C08959=1014.055,42.022,-115.275,165.854,58.897,160.635
C08960=1014.061,42.301,-115.291,165.856,58.886,160.634
C08961=1014.066,42.582,-115.308,165.859,58.876,160.633
C08962=1014.071,42.863,-115.324,165.862,58.866,160.631
C08963=1014.075,43.112,-115.338,165.863,58.857,160.630
C08964=1014.080,43.362,-115.352,165.865,58.848,160.628
C08965=1014.085,43.611,-115.367,165.867,58.838,160.627
C08966=1014.089,43.860,-115.381,165.869,58.829,160.626
C08967=1014.094,44.110,-115.396,165.872,58.820,160.625
C08968=1014.099,44.360,-115.410,165.875,58.810,160.624
C08969=1014.103,44.609,-115.424,165.877,58.800,160.622
C08970=1014.108,44.859,-115.440,165.879,58.791,160.621
C08971=1014.113,45.108,-115.454,165.881,58.782,160.620
C08972=1014.117,45.358,-115.468,165.883,58.773,160.619
C08973=1014.121,45.608,-115.483,165.885,58.763,160.617
C08974=1014.126,45.857,-115.497,165.887,58.754,160.616
C08975=1014.131,46.106,-115.512,165.890,58.745,160.615
C08976=1014.135,46.356,-115.526,165.892,58.735,160.613
C08977=1014.140,46.606,-115.541,165.894,58.726,160.612
C08978=1014.144,46.855,-115.555,165.896,58.716,160.611
C08979=1014.149,47.104,-115.570,165.898,58.707,160.610
C08980=1014.154,47.354,-115.585,165.900,58.697,160.608
C08981=1014.158,47.603,-115.599,165.902,58.688,160.607
C08982=1014.163,47.853,-115.613,165.905,58.678,160.606
C08983=1014.168,48.102,-115.628,165.907,58.668,160.604
C08984=1014.173,48.352,-115.643,165.910,58.659,160.603
C08985=1014.177,48.601,-115.657,165.911,58.650,160.602
C08986=1014.182,48.851,-115.671,165.914,58.641,160.601
C08987=1014.187,49.101,-115.686,165.916,58.631,160.599
C08988=1014.191,49.351,-115.701,165.917,58.621,160.598
C08989=1014.196,49.600,-115.715,165.921,58.612,160.597
C08990=1014.200,49.850,-115.730,165.923,58.602,160.596
C08991=1014.205,50.099,-115.745,165.924,58.592,160.594
C08992=1014.210,50.349,-115.759,165.927,58.583,160.593
C08993=1014.214,50.598,-115.773,165.929,58.573,160.592
C08994=1014.219,50.847,-115.788,165.931,58.564,160.590
C08995=1014.224,51.097,-115.803,165.934,58.554,160.589
C08996=1014.228,51.347,-115.818,165.936,58.544,160.588
C08997=1014.232,51.596,-115.833,165.938,58.535,160.586
C08998=1014.237,51.846,-115.847,165.940,58.525,160.585
C08999=1014.242,52.096,-115.862,165.943,58.515,160.584
C09000=1014.247,52.345,-115.877,165.945,58.506,160.583
C09001=1014.251,52.594,-115.891,165.947,58.496,160.581
C09002=1014.256,52.844,-115.905,165.949,58.486,160.580
C09003=1014.261,53.093,-115.921,165.952,58.477,160.579
C09004=1014.266,53.343,-115.935,165.954,58.467,160.577
C09005=1014.270,53.593,-115.949,165.956,58.457,160.576
C09006=1014.275,53.842,-115.964,165.958,58.448,160.574
C09007=1014.279,54.091,-115.979,165.961,58.437,160.573
C09008=1014.285,54.341,-115.994,165.962,58.428,160.572
C09009=1014.289,54.591,-116.008,165.964,58.418,160.570
C09010=1014.294,54.841,-116.023,165.968,58.409,160.569
C09011=1014.299,55.090,-116.038,165.970,58.399,160.568
C09012=1014.303,55.339,-116.052,165.971,58.389,160.567
C09013=1014.308,55.588,-116.067,165.974,58.379,160.565
C09014=1014.313,55.838,-116.082,165.976,58.369,160.564
C09015=1014.318,56.088,-116.096,165.978,58.359,160.562
C09016=1014.323,56.337,-116.111,165.981,58.349,160.561
C09017=1014.327,56.587,-116.126,165.983,58.340,160.560
C09018=1014.332,56.836,-116.141,165.985,58.330,160.558
C09019=1014.337,57.086,-116.155,165.988,58.320,160.557
C09020=1014.342,57.335,-116.170,165.990,58.310,160.556
C09021=1014.346,57.585,-116.185,165.993,58.300,160.555
C09022=1014.351,57.835,-116.199,165.995,58.290,160.553
C09023=1014.357,58.115,-116.216,165.997,58.279,160.552
C09024=1014.362,58.394,-116.233,166.000,58.268,160.550
C09025=1014.367,58.675,-116.249,166.003,58.257,160.549
C09026=1014.372,58.956,-116.266,166.004,58.245,160.547
C09027=1014.377,59.205,-116.280,166.007,58.235,160.546
C09028=1014.382,59.455,-116.296,166.009,58.226,160.544
C09029=1014.387,59.705,-116.310,166.011,58.216,160.543
C09030=1014.392,59.954,-116.325,166.014,58.206,160.542
C09031=1014.397,60.204,-116.340,166.016,58.196,160.540
C09032=1014.401,60.452,-116.355,166.019,58.186,160.539
C09033=1014.406,60.702,-116.369,166.020,58.176,160.537
C09034=1014.411,60.951,-116.384,166.023,58.165,160.536
C09035=1014.416,61.201,-116.399,166.025,58.156,160.535
C09036=1014.421,61.451,-116.414,166.028,58.146,160.533
C09037=1014.426,61.700,-116.429,166.030,58.136,160.532
C09038=1014.430,61.950,-116.443,166.033,58.126,160.531
C09039=1014.436,62.199,-116.459,166.034,58.115,160.529
C09040=1014.440,62.449,-116.473,166.037,58.105,160.528
C09041=1014.445,62.698,-116.488,166.039,58.096,160.526
C09042=1014.449,62.948,-116.503,166.042,58.085,160.525
C09043=1014.454,63.198,-116.518,166.044,58.076,160.524
C09044=1014.459,63.447,-116.534,166.046,58.066,160.522
C09045=1014.464,63.696,-116.549,166.049,58.056,160.521
C09046=1014.468,63.946,-116.564,166.051,58.046,160.520
C09047=1014.473,64.196,-116.579,166.054,58.036,160.519
C09048=1014.478,64.445,-116.595,166.056,58.026,160.517
C09049=1014.482,64.694,-116.610,166.058,58.016,160.516
C09050=1014.487,64.944,-116.624,166.061,58.006,160.514
C09051=1014.491,65.193,-116.640,166.062,57.996,160.513
C09052=1014.496,65.442,-116.655,166.066,57.986,160.512
C09053=1014.501,65.692,-116.670,166.067,57.977,160.510
C09054=1014.506,65.941,-116.686,166.069,57.967,160.509
C09055=1014.510,66.191,-116.700,166.072,57.956,160.507
C09056=1014.515,66.441,-116.716,166.074,57.946,160.506
C09057=1014.520,66.690,-116.731,166.077,57.936,160.505
C09058=1014.525,66.939,-116.747,166.079,57.927,160.503
C09059=1014.529,67.189,-116.762,166.082,57.917,160.502
C09060=1014.534,67.438,-116.778,166.084,57.907,160.501
C09061=1014.538,67.688,-116.793,166.086,57.896,160.499
C09062=1014.543,67.938,-116.808,166.088,57.886,160.498
C09063=1014.548,68.187,-116.823,166.090,57.877,160.497
C09064=1014.553,68.436,-116.839,166.093,57.867,160.495
C09065=1014.557,68.686,-116.854,166.095,57.857,160.494
C09066=1014.562,68.935,-116.870,166.098,57.846,160.492
C09067=1014.566,69.185,-116.885,166.100,57.837,160.491
C09068=1014.571,69.434,-116.901,166.103,57.827,160.490
C09069=1014.576,69.684,-116.916,166.105,57.817,160.488
C09070=1014.581,69.934,-116.932,166.108,57.807,160.487
C09071=1014.585,70.183,-116.948,166.109,57.796,160.486
C09072=1014.591,70.433,-116.963,166.111,57.787,160.484
C09073=1014.595,70.682,-116.979,166.115,57.777,160.483
C09074=1014.599,70.932,-116.994,166.117,57.767,160.482
C09075=1014.604,71.181,-117.010,166.119,57.756,160.480
C09076=1014.608,71.431,-117.025,166.121,57.747,160.479
C09077=1014.614,71.680,-117.040,166.124,57.737,160.478
C09078=1014.618,71.929,-117.056,166.126,57.727,160.476
C09079=1014.623,72.179,-117.071,166.129,57.716,160.475
C09080=1014.627,72.428,-117.087,166.131,57.707,160.473
C09081=1014.631,72.678,-117.103,166.134,57.697,160.472
C09082=1014.637,72.927,-117.118,166.136,57.687,160.471
C09083=1014.641,73.177,-117.134,166.138,57.676,160.469
C09084=1014.646,73.426,-117.149,166.140,57.666,160.468
C09085=1014.650,73.675,-117.166,166.144,57.656,160.467
C09086=1014.655,73.925,-117.182,166.145,57.646,160.465
C09087=1014.661,74.206,-117.199,166.149,57.635,160.464
C09088=1014.666,74.486,-117.216,166.150,57.623,160.462
C09089=1014.671,74.766,-117.234,166.154,57.612,160.461
C09090=1014.676,75.046,-117.252,166.156,57.601,160.459
C09091=1014.681,75.295,-117.267,166.159,57.591,160.458
C09092=1014.686,75.545,-117.282,166.161,57.580,160.456
C09093=1014.691,75.795,-117.299,166.164,57.570,160.455
C09094=1014.696,76.045,-117.314,166.167,57.560,160.454
C09095=1014.700,76.294,-117.330,166.168,57.550,160.452
C09096=1014.705,76.543,-117.346,166.171,57.540,160.451
C09097=1014.709,76.793,-117.362,166.173,57.530,160.449
C09098=1014.714,77.042,-117.377,166.176,57.519,160.448
C09099=1014.718,77.292,-117.393,166.178,57.510,160.447
C09100=1014.723,77.541,-117.410,166.181,57.499,160.445
C09101=1014.728,77.791,-117.425,166.183,57.490,160.444
C09102=1014.732,78.040,-117.441,166.186,57.480,160.443
C09103=1014.737,78.289,-117.458,166.187,57.469,160.441
C09104=1014.741,78.539,-117.473,166.191,57.459,160.440
C09105=1014.746,78.788,-117.489,166.193,57.450,160.438
C09106=1014.751,79.038,-117.505,166.195,57.439,160.437
C09107=1014.755,79.287,-117.521,166.197,57.429,160.435
C09108=1014.760,79.537,-117.537,166.201,57.419,160.434
C09109=1014.764,79.786,-117.553,166.202,57.409,160.433
C09110=1014.769,80.035,-117.569,166.205,57.399,160.431
C09111=1014.773,80.285,-117.585,166.207,57.389,160.430
C09112=1014.778,80.535,-117.602,166.210,57.379,160.429
C09113=1014.783,80.784,-117.617,166.212,57.369,160.427
C09114=1014.788,81.033,-117.633,166.215,57.358,160.426
C09115=1014.792,81.283,-117.649,166.217,57.349,160.424
C09116=1014.796,81.532,-117.665,166.219,57.338,160.423
C09117=1014.802,81.782,-117.682,166.223,57.328,160.422
C09118=1014.806,82.031,-117.698,166.224,57.318,160.420
C09119=1014.811,82.280,-117.714,166.227,57.308,160.419
C09120=1014.815,82.530,-117.730,166.229,57.297,160.417
C09121=1014.819,82.779,-117.746,166.232,57.287,160.416
C09122=1014.825,83.029,-117.762,166.235,57.277,160.415
C09123=1014.829,83.278,-117.778,166.237,57.267,160.413
C09124=1014.834,83.527,-117.794,166.240,57.256,160.412
C09125=1014.838,83.777,-117.810,166.242,57.247,160.411
C09126=1014.844,84.027,-117.827,166.244,57.236,160.409
C09127=1014.848,84.276,-117.843,166.248,57.226,160.408
C09128=1014.852,84.526,-117.858,166.249,57.216,160.406
C09129=1014.857,84.775,-117.875,166.252,57.206,160.405
C09130=1014.862,85.025,-117.891,166.255,57.195,160.404
C09131=1014.867,85.274,-117.907,166.257,57.185,160.402
C09132=1014.871,85.523,-117.923,166.260,57.175,160.401
C09133=1014.876,85.772,-117.939,166.262,57.164,160.399
C09134=1014.881,86.022,-117.955,166.265,57.155,160.398
C09135=1014.886,86.271,-117.972,166.267,57.144,160.397
C09136=1014.890,86.521,-117.987,166.270,57.133,160.395
C09137=1014.895,86.771,-118.004,166.272,57.124,160.394
C09138=1014.899,87.020,-118.020,166.275,57.113,160.392
C09139=1014.904,87.269,-118.037,166.277,57.102,160.391
C09140=1014.909,87.518,-118.052,166.280,57.093,160.390
C09141=1014.914,87.768,-118.069,166.282,57.082,160.388
C09142=1014.919,88.018,-118.084,166.285,57.071,160.387
C09143=1014.923,88.267,-118.101,166.288,57.061,160.386
C09144=1014.928,88.517,-118.117,166.290,57.051,160.384
C09145=1014.933,88.766,-118.134,166.292,57.041,160.382
C09146=1014.937,89.015,-118.150,166.296,57.031,160.381
C09147=1014.942,89.265,-118.166,166.297,57.020,160.380
C09148=1014.946,89.514,-118.183,166.301,57.010,160.378
C09149=1014.951,89.763,-118.200,166.302,57.000,160.377
C09150=1014.956,90.013,-118.217,166.306,56.990,160.376
C09151=1014.960,90.294,-118.234,166.309,56.978,160.374
C09152=1014.966,90.575,-118.253,166.311,56.967,160.372
C09153=1014.970,90.855,-118.272,166.314,56.955,160.371
C09154=1014.976,91.135,-118.290,166.317,56.944,160.369
C09155=1014.980,91.384,-118.307,166.319,56.934,160.368
C09156=1014.985,91.634,-118.324,166.323,56.924,160.367
C09157=1014.990,91.884,-118.340,166.324,56.914,160.365
C09158=1014.994,92.133,-118.356,166.327,56.903,160.364
C09159=1015.000,92.382,-118.373,166.330,56.893,160.363
C09160=1015.003,92.631,-118.390,166.332,56.883,160.361
C09161=1015.008,92.880,-118.407,166.335,56.872,160.360
C09162=1015.013,93.131,-118.423,166.338,56.862,160.358
C09163=1015.018,93.380,-118.440,166.340,56.852,160.357
C09164=1015.022,93.630,-118.457,166.343,56.841,160.355
C09165=1015.027,93.879,-118.473,166.346,56.831,160.354
C09166=1015.031,94.128,-118.490,166.348,56.821,160.353
C09167=1015.036,94.378,-118.506,166.350,56.811,160.351
C09168=1015.041,94.627,-118.523,166.354,56.801,160.350
C09169=1015.045,94.876,-118.540,166.355,56.790,160.348
C09170=1015.050,95.126,-118.556,166.358,56.780,160.347
C09171=1015.055,95.375,-118.573,166.361,56.770,160.346
C09172=1015.060,95.624,-118.590,166.364,56.759,160.344
C09173=1015.064,95.873,-118.606,166.366,56.749,160.343
C09174=1015.069,96.124,-118.623,166.369,56.738,160.341
C09175=1015.073,96.373,-118.640,166.372,56.728,160.340
C09176=1015.078,96.622,-118.656,166.375,56.718,160.339
C09177=1015.083,96.871,-118.673,166.376,56.708,160.337
C09178=1015.087,97.121,-118.690,166.379,56.697,160.336
C09179=1015.092,97.370,-118.707,166.382,56.686,160.334
C09180=1015.097,97.619,-118.723,166.385,56.676,160.333
C09181=1015.102,97.869,-118.740,166.387,56.666,160.332
C09182=1015.106,98.118,-118.757,166.390,56.656,160.330
C09183=1015.110,98.367,-118.774,166.393,56.645,160.329
C09184=1015.115,98.618,-118.790,166.395,56.634,160.327
C09185=1015.120,98.866,-118.806,166.399,56.625,160.326
C09186=1015.124,99.116,-118.824,166.401,56.614,160.325
C09187=1015.129,99.365,-118.841,166.403,56.604,160.323
C09188=1015.134,99.615,-118.858,166.407,56.594,160.322
C09189=1015.138,99.864,-118.875,166.408,56.584,160.320
C09190=1015.143,100.114,-118.892,166.411,56.573,160.319
C09191=1015.147,100.363,-118.909,166.415,56.563,160.318
C09192=1015.152,100.613,-118.926,166.416,56.553,160.316
C09193=1015.157,100.862,-118.943,166.419,56.542,160.315
C09194=1015.161,101.112,-118.960,166.422,56.532,160.313
C09195=1015.166,101.360,-118.977,166.424,56.522,160.312
C09196=1015.170,101.610,-118.995,166.427,56.512,160.311
C09197=1015.175,101.859,-119.011,166.430,56.501,160.309
C09198=1015.179,102.109,-119.029,166.433,56.491,160.308
C09199=1015.184,102.358,-119.045,166.435,56.481,160.307
C09200=1015.189,102.608,-119.063,166.438,56.471,160.305
C09201=1015.193,102.857,-119.079,166.441,56.460,160.304
C09202=1015.198,103.106,-119.097,166.444,56.449,160.302
C09203=1015.203,103.355,-119.114,166.446,56.440,160.301
C09204=1015.207,103.605,-119.131,166.449,56.429,160.300
C09205=1015.212,103.854,-119.148,166.452,56.419,160.298
C09206=1015.216,104.104,-119.165,166.455,56.408,160.297
C09207=1015.221,104.352,-119.182,166.457,56.399,160.296
C09208=1015.226,104.602,-119.200,166.460,56.388,160.294
C09209=1015.229,104.851,-119.217,166.463,56.378,160.293
C09210=1015.235,105.101,-119.234,166.466,56.367,160.291
C09211=1015.239,105.350,-119.252,166.467,56.357,160.290
C09212=1015.244,105.599,-119.268,166.470,56.346,160.288
C09213=1015.248,105.849,-119.286,166.474,56.336,160.287
C09214=1015.253,106.098,-119.302,166.477,56.326,160.286
C09215=1015.259,106.379,-119.322,166.480,56.314,160.284
C09216=1015.263,106.660,-119.342,166.482,56.302,160.282
C09217=1015.269,106.940,-119.361,166.485,56.290,160.281
C09218=1015.275,107.222,-119.380,166.488,56.279,160.279
C09219=1015.279,107.471,-119.398,166.491,56.268,160.278
C09220=1015.284,107.720,-119.415,166.494,56.258,160.277
C09221=1015.288,107.970,-119.432,166.498,56.248,160.275
C09222=1015.293,108.219,-119.449,166.500,56.238,160.274
C09223=1015.298,108.469,-119.467,166.502,56.227,160.272
C09224=1015.302,108.717,-119.483,166.505,56.217,160.271
C09225=1015.307,108.967,-119.501,166.508,56.206,160.270
C09226=1015.311,109.216,-119.518,166.511,56.196,160.268
C09227=1015.316,109.466,-119.535,166.514,56.185,160.267
C09228=1015.321,109.715,-119.553,166.516,56.175,160.265
C09229=1015.325,109.964,-119.570,166.519,56.164,160.264
C09230=1015.330,110.213,-119.588,166.522,56.155,160.263
C09231=1015.335,110.463,-119.605,166.525,56.144,160.261
C09232=1015.339,110.713,-119.623,166.528,56.133,160.260
C09233=1015.344,110.962,-119.641,166.530,56.123,160.258
C09234=1015.348,111.211,-119.657,166.533,56.113,160.257
C09235=1015.353,111.460,-119.675,166.536,56.102,160.256
C09236=1015.357,111.710,-119.693,166.539,56.092,160.254
C09237=1015.362,111.959,-119.711,166.542,56.081,160.253
C09238=1015.366,112.209,-119.728,166.544,56.072,160.252
C09239=1015.371,112.458,-119.746,166.547,56.061,160.250
C09240=1015.375,112.707,-119.764,166.550,56.051,160.249
C09241=1015.380,112.957,-119.781,166.553,56.040,160.247
C09242=1015.384,113.206,-119.800,166.556,56.031,160.246
C09243=1015.389,113.455,-119.817,166.558,56.020,160.245
C09244=1015.393,113.705,-119.835,166.561,56.010,160.243
C09245=1015.398,113.954,-119.853,166.564,55.999,160.242
C09246=1015.402,114.203,-119.871,166.567,55.990,160.241
C09247=1015.406,114.453,-119.888,166.570,55.980,160.239
C09248=1015.411,114.702,-119.906,166.573,55.969,160.238
C09249=1015.415,114.951,-119.924,166.576,55.959,160.237
C09250=1015.420,115.201,-119.942,166.578,55.949,160.235
C09251=1015.425,115.450,-119.960,166.581,55.939,160.234
C09252=1015.429,115.700,-119.978,166.584,55.928,160.232
C09253=1015.434,115.948,-119.996,166.587,55.918,160.231
C09254=1015.438,116.198,-120.013,166.590,55.907,160.230
C09255=1015.443,116.447,-120.031,166.592,55.897,160.228
C09256=1015.447,116.696,-120.049,166.596,55.887,160.227
C09257=1015.452,116.945,-120.067,166.599,55.877,160.226
C09258=1015.456,117.195,-120.085,166.602,55.866,160.224
C09259=1015.460,117.416,-120.100,166.604,55.857,160.223
C09260=1015.464,117.636,-120.117,166.607,55.848,160.222
C09261=1015.469,117.857,-120.133,166.610,55.839,160.221
C09262=1015.473,118.078,-120.148,166.611,55.830,160.219
C09263=1015.477,118.298,-120.164,166.614,55.821,160.218
C09264=1015.481,118.519,-120.179,166.617,55.812,160.217
C09265=1015.484,118.740,-120.196,166.619,55.803,160.216
C09266=1015.488,118.961,-120.212,166.622,55.793,160.214
C09267=1015.493,119.210,-120.230,166.625,55.783,160.213
C09268=1015.497,119.459,-120.247,166.628,55.773,160.212
C09269=1015.502,119.708,-120.266,166.631,55.762,160.210
C09270=1015.507,119.957,-120.284,166.634,55.752,160.209
C09271=1015.512,120.207,-120.302,166.636,55.742,160.208
C09272=1015.516,120.456,-120.319,166.639,55.732,160.206
C09273=1015.520,120.705,-120.337,166.642,55.721,160.205
C09274=1015.525,120.955,-120.355,166.645,55.711,160.204
C09275=1015.530,121.204,-120.374,166.648,55.700,160.202
C09276=1015.535,121.453,-120.392,166.651,55.690,160.201
C09277=1015.539,121.702,-120.409,166.654,55.680,160.199
C09278=1015.543,121.952,-120.427,166.657,55.669,160.198
C09279=1015.550,122.290,-120.452,166.660,55.655,160.196
C09280=1015.556,122.628,-120.476,166.665,55.641,160.194
C09281=1015.563,122.967,-120.501,166.669,55.627,160.192
C09282=1015.568,123.305,-120.525,166.674,55.613,160.191
C09283=1015.573,123.554,-120.543,166.677,55.602,160.189
C09284=1015.578,123.804,-120.561,166.680,55.592,160.188
C09285=1015.583,124.053,-120.580,166.682,55.582,160.186
C09286=1015.588,124.302,-120.598,166.685,55.571,160.185
C09287=1015.592,124.551,-120.616,166.688,55.561,160.184
C09288=1015.597,124.800,-120.634,166.691,55.551,160.182
C09289=1015.601,125.050,-120.652,166.694,55.540,160.181
C09290=1015.606,125.299,-120.670,166.697,55.530,160.180
C09291=1015.611,125.549,-120.687,166.700,55.519,160.178
C09292=1015.615,125.798,-120.706,166.703,55.509,160.177
C09293=1015.620,126.048,-120.724,166.706,55.498,160.175
C09294=1015.625,126.297,-120.742,166.709,55.487,160.174
C09295=1015.629,126.546,-120.760,166.712,55.477,160.173
C09296=1015.634,126.795,-120.778,166.715,55.466,160.171
C09297=1015.639,127.044,-120.796,166.718,55.456,160.170
C09298=1015.643,127.294,-120.814,166.722,55.446,160.168
C09299=1015.648,127.543,-120.832,166.725,55.435,160.167
C09300=1015.653,127.792,-120.851,166.728,55.425,160.166
C09301=1015.658,128.042,-120.869,166.731,55.414,160.164
C09302=1015.663,128.291,-120.887,166.734,55.404,160.163
C09303=1015.667,128.540,-120.905,166.737,55.394,160.162
C09304=1015.671,128.790,-120.924,166.740,55.383,160.160
C09305=1015.676,129.039,-120.943,166.743,55.372,160.159
C09306=1015.681,129.288,-120.961,166.746,55.362,160.157
C09307=1015.685,129.537,-120.979,166.749,55.351,160.156
C09308=1015.690,129.786,-120.997,166.752,55.341,160.155
C09309=1015.694,130.036,-121.016,166.755,55.330,160.153
C09310=1015.700,130.286,-121.034,166.758,55.320,160.152
C09311=1015.704,130.535,-121.052,166.762,55.310,160.151
C09312=1015.708,130.784,-121.071,166.765,55.300,160.149
C09313=1015.713,131.033,-121.089,166.768,55.290,160.148
C09314=1015.717,131.283,-121.108,166.772,55.279,160.147
C09315=1015.722,131.531,-121.127,166.775,55.269,160.145
C09316=1015.727,131.781,-121.145,166.777,55.259,160.144
C09317=1015.731,132.030,-121.164,166.780,55.249,160.143
C09318=1015.736,132.280,-121.182,166.783,55.238,160.141
C09319=1015.740,132.529,-121.202,166.786,55.228,160.140
C09320=1015.745,132.778,-121.220,166.789,55.217,160.138
C09321=1015.750,133.027,-121.238,166.793,55.207,160.137
C09322=1015.754,133.276,-121.257,166.796,55.197,160.136
C09323=1015.759,133.526,-121.276,166.799,55.186,160.134
C09324=1015.763,133.775,-121.294,166.802,55.176,160.133
C09325=1015.768,134.024,-121.313,166.805,55.166,160.132
C09326=1015.773,134.274,-121.331,166.808,55.155,160.130
C09327=1015.777,134.523,-121.350,166.812,55.145,160.129
C09328=1015.782,134.772,-121.369,166.815,55.135,160.128
C09329=1015.786,135.021,-121.387,166.818,55.124,160.126
C09330=1015.791,135.270,-121.407,166.821,55.114,160.125
C09331=1015.796,135.520,-121.425,166.824,55.103,160.124
C09332=1015.800,135.769,-121.444,166.828,55.093,160.122
C09333=1015.805,136.018,-121.462,166.831,55.083,160.121
C09334=1015.809,136.268,-121.481,166.834,55.072,160.120
C09335=1015.814,136.516,-121.500,166.837,55.062,160.118
C09336=1015.818,136.766,-121.519,166.840,55.052,160.117
C09337=1015.823,137.015,-121.538,166.844,55.041,160.116
C09338=1015.828,137.265,-121.557,166.847,55.031,160.114
C09339=1015.833,137.514,-121.576,166.850,55.021,160.113
C09340=1015.837,137.764,-121.594,166.853,55.010,160.112
C09341=1015.842,138.012,-121.613,166.856,55.000,160.110
C09342=1015.846,138.262,-121.632,166.860,54.990,160.109
C09343=1015.851,138.543,-121.654,166.863,54.978,160.107
C09344=1015.856,138.823,-121.675,166.867,54.967,160.106
C09345=1015.861,139.104,-121.696,166.871,54.955,160.105
C09346=1015.866,139.385,-121.718,166.874,54.943,160.103
C09347=1015.871,139.634,-121.737,166.877,54.933,160.102
C09348=1015.875,139.884,-121.756,166.881,54.923,160.100
C09349=1015.879,140.133,-121.775,166.884,54.913,160.099
C09350=1015.885,140.382,-121.795,166.888,54.903,160.098
C09351=1015.889,140.632,-121.813,166.891,54.892,160.096
C09352=1015.894,140.881,-121.833,166.894,54.882,160.095
C09353=1015.899,141.129,-121.852,166.897,54.872,160.094
C09354=1015.903,141.379,-121.870,166.901,54.861,160.092
C09355=1015.907,141.628,-121.890,166.904,54.851,160.091
C09356=1015.912,141.877,-121.909,166.907,54.841,160.090
C09357=1015.916,142.127,-121.928,166.910,54.831,160.088
C09358=1015.921,142.376,-121.947,166.914,54.820,160.087
C09359=1015.926,142.625,-121.966,166.917,54.810,160.086
C09360=1015.930,142.875,-121.985,166.920,54.800,160.084
C09361=1015.935,143.123,-122.004,166.923,54.789,160.083
C09362=1015.940,143.373,-122.023,166.927,54.779,160.082
C09363=1015.944,143.622,-122.043,166.930,54.769,160.080
C09364=1015.949,143.872,-122.061,166.933,54.759,160.079
C09365=1015.954,144.121,-122.081,166.937,54.748,160.078
C09366=1015.958,144.370,-122.100,166.940,54.738,160.076
C09367=1015.963,144.618,-122.119,166.943,54.728,160.075
C09368=1015.967,144.868,-122.138,166.946,54.717,160.074
C09369=1015.972,145.117,-122.157,166.950,54.707,160.072
C09370=1015.977,145.367,-122.177,166.953,54.697,160.071
C09371=1015.982,145.616,-122.196,166.956,54.687,160.070
C09372=1015.986,145.865,-122.216,166.960,54.676,160.068
C09373=1015.990,146.114,-122.235,166.963,54.666,160.067
C09374=1015.995,146.363,-122.255,166.966,54.656,160.066
C09375=1015.999,146.613,-122.274,166.970,54.645,160.064
C09376=1016.004,146.862,-122.293,166.973,54.635,160.063
C09377=1016.008,147.111,-122.313,166.976,54.625,160.062
C09378=1016.013,147.360,-122.331,166.979,54.615,160.061
C09379=1016.018,147.610,-122.351,166.984,54.604,160.059
C09380=1016.022,147.859,-122.371,166.987,54.594,160.058
C09381=1016.027,148.108,-122.390,166.990,54.583,160.057
C09382=1016.031,148.357,-122.410,166.994,54.573,160.055
C09383=1016.036,148.607,-122.430,166.997,54.563,160.054
C09384=1016.040,148.856,-122.449,167.000,54.553,160.053
C09385=1016.045,149.105,-122.469,167.004,54.543,160.052
C09386=1016.049,149.354,-122.488,167.008,54.533,160.050
C09387=1016.054,149.603,-122.508,167.011,54.523,160.049
C09388=1016.058,149.852,-122.527,167.014,54.512,160.048
C09389=1016.063,150.101,-122.547,167.018,54.502,160.046
C09390=1016.068,150.351,-122.567,167.021,54.492,160.045
C09391=1016.072,150.600,-122.586,167.024,54.482,160.044
C09392=1016.077,150.849,-122.605,167.028,54.472,160.042
C09393=1016.082,151.097,-122.625,167.031,54.461,160.041
C09394=1016.087,151.347,-122.645,167.034,54.451,160.040
C09395=1016.091,151.596,-122.664,167.038,54.441,160.038
C09396=1016.095,151.845,-122.684,167.041,54.431,160.037
C09397=1016.100,152.095,-122.704,167.045,54.420,160.036
C09398=1016.105,152.344,-122.723,167.049,54.410,160.035
C09399=1016.109,152.593,-122.743,167.052,54.400,160.033
C09400=1016.114,152.843,-122.763,167.056,54.389,160.032
C09401=1016.119,153.091,-122.783,167.059,54.379,160.031
C09402=1016.123,153.340,-122.802,167.062,54.369,160.029
C09403=1016.127,153.590,-122.823,167.066,54.359,160.028
C09404=1016.132,153.839,-122.842,167.070,54.349,160.027
C09405=1016.136,154.088,-122.862,167.073,54.339,160.026
C09406=1016.141,154.338,-122.882,167.076,54.329,160.024
C09407=1016.146,154.618,-122.904,167.080,54.317,160.023
C09408=1016.152,154.899,-122.927,167.084,54.305,160.021
C09409=1016.157,155.180,-122.949,167.089,54.294,160.020
C09410=1016.162,155.460,-122.971,167.093,54.282,160.019
C09411=1016.166,155.710,-122.992,167.096,54.272,160.017
C09412=1016.171,155.959,-123.011,167.099,54.262,160.016
C09413=1016.176,156.209,-123.031,167.103,54.252,160.015
C09414=1016.180,156.457,-123.051,167.106,54.242,160.013
C09415=1016.185,156.706,-123.071,167.110,54.231,160.012
C09416=1016.189,156.956,-123.091,167.113,54.221,160.011
C09417=1016.194,157.204,-123.111,167.118,54.211,160.010
C09418=1016.199,157.454,-123.131,167.121,54.201,160.008
C09419=1016.203,157.703,-123.150,167.125,54.191,160.007
C09420=1016.207,157.952,-123.171,167.128,54.181,160.006
C09421=1016.212,158.202,-123.191,167.132,54.171,160.004
C09422=1016.217,158.451,-123.210,167.135,54.160,160.003
C09423=1016.222,158.700,-123.231,167.139,54.150,160.002
C09424=1016.226,158.948,-123.251,167.142,54.140,160.001
C09425=1016.231,159.198,-123.271,167.146,54.131,159.999
C09426=1016.235,159.447,-123.292,167.149,54.121,159.998
C09427=1016.238,159.696,-123.312,167.153,54.110,159.997
C09428=1016.244,159.945,-123.333,167.157,54.101,159.996
C09429=1016.247,160.194,-123.354,167.160,54.091,159.994
C09430=1016.252,160.444,-123.373,167.164,54.081,159.993
C09431=1016.256,160.693,-123.394,167.167,54.070,159.992
C09432=1016.261,160.942,-123.415,167.171,54.061,159.991
C09433=1016.265,161.191,-123.435,167.174,54.051,159.990
C09434=1016.270,161.441,-123.456,167.178,54.041,159.988
C09435=1016.274,161.689,-123.476,167.181,54.030,159.987
C09436=1016.279,161.938,-123.497,167.185,54.021,159.986
C09437=1016.283,162.187,-123.517,167.190,54.010,159.985
C09438=1016.287,162.436,-123.537,167.193,54.000,159.983
C09439=1016.292,162.686,-123.559,167.197,53.991,159.982
C09440=1016.296,162.935,-123.578,167.201,53.981,159.981
C09441=1016.301,163.184,-123.599,167.204,53.971,159.980
C09442=1016.306,163.433,-123.620,167.208,53.960,159.978
C09443=1016.310,163.682,-123.641,167.211,53.951,159.977
C09444=1016.314,163.932,-123.661,167.215,53.941,159.976
C09445=1016.319,164.180,-123.681,167.218,53.931,159.975
C09446=1016.323,164.430,-123.702,167.222,53.921,159.973
C09447=1016.328,164.678,-123.723,167.226,53.911,159.972
C09448=1016.332,164.928,-123.744,167.229,53.901,159.971
C09449=1016.337,165.177,-123.763,167.234,53.891,159.970
C09450=1016.341,165.426,-123.784,167.237,53.880,159.969
C09451=1016.345,165.675,-123.805,167.241,53.870,159.967
C09452=1016.350,165.924,-123.826,167.245,53.861,159.966
C09453=1016.354,166.173,-123.846,167.248,53.851,159.965
C09454=1016.359,166.422,-123.867,167.252,53.841,159.964
C09455=1016.364,166.672,-123.887,167.255,53.831,159.962
C09456=1016.368,166.921,-123.908,167.259,53.821,159.961
C09457=1016.373,167.170,-123.929,167.264,53.811,159.960
C09458=1016.377,167.419,-123.950,167.267,53.801,159.959
C09459=1016.382,167.668,-123.970,167.271,53.790,159.957
C09460=1016.387,167.917,-123.991,167.274,53.780,159.956
C09461=1016.390,168.166,-124.012,167.278,53.771,159.955
C09462=1016.396,168.415,-124.033,167.282,53.761,159.954
C09463=1016.400,168.664,-124.054,167.286,53.750,159.953
C09464=1016.405,168.913,-124.074,167.290,53.740,159.951
C09465=1016.409,169.163,-124.094,167.294,53.730,159.950
C09466=1016.413,169.412,-124.115,167.298,53.721,159.949
C09467=1016.418,169.661,-124.136,167.301,53.711,159.948
C09468=1016.423,169.910,-124.157,167.306,53.700,159.947
C09469=1016.427,170.159,-124.177,167.309,53.690,159.945
C09470=1016.432,170.408,-124.198,167.313,53.680,159.944
C09471=1016.437,170.688,-124.222,167.317,53.669,159.943
C09472=1016.443,170.969,-124.245,167.321,53.658,159.941
C09473=1016.447,171.250,-124.268,167.326,53.646,159.940
C09474=1016.453,171.530,-124.293,167.330,53.635,159.938
C09475=1016.458,171.779,-124.313,167.334,53.625,159.937
C09476=1016.462,172.028,-124.334,167.339,53.615,159.936
C09477=1016.467,172.277,-124.355,167.342,53.605,159.935
C09478=1016.472,172.527,-124.376,167.346,53.595,159.934
C09479=1016.476,172.775,-124.397,167.349,53.585,159.932
C09480=1016.481,173.024,-124.417,167.354,53.575,159.931
C09481=1016.486,173.274,-124.438,167.358,53.564,159.930
C09482=1016.490,173.522,-124.458,167.362,53.555,159.929
C09483=1016.495,173.772,-124.480,167.365,53.545,159.928
C09484=1016.499,174.021,-124.501,167.370,53.535,159.926
C09485=1016.505,174.270,-124.521,167.373,53.525,159.925
C09486=1016.509,174.520,-124.542,167.377,53.515,159.924
C09487=1016.513,174.769,-124.563,167.382,53.505,159.923
C09488=1016.519,175.017,-124.584,167.386,53.495,159.922
C09489=1016.523,175.266,-124.606,167.389,53.485,159.920
C09490=1016.528,175.516,-124.626,167.393,53.475,159.919
C09491=1016.532,175.764,-124.647,167.397,53.464,159.918
C09492=1016.537,176.014,-124.668,167.401,53.454,159.917
C09493=1016.542,176.263,-124.689,167.405,53.444,159.915
C09494=1016.547,176.512,-124.711,167.410,53.434,159.914
C09495=1016.552,176.761,-124.731,167.413,53.424,159.913
C09496=1016.557,177.010,-124.752,167.417,53.414,159.912
C09497=1016.561,177.259,-124.773,167.422,53.404,159.911
C09498=1016.566,177.508,-124.794,167.425,53.394,159.909
C09499=1016.571,177.757,-124.815,167.429,53.384,159.908
C09500=1016.576,178.006,-124.836,167.434,53.374,159.907
C09501=1016.580,178.255,-124.857,167.438,53.364,159.906
C09502=1016.585,178.505,-124.878,167.442,53.354,159.905
C09503=1016.590,178.753,-124.900,167.446,53.344,159.903
C09504=1016.594,179.002,-124.920,167.449,53.334,159.902
C09505=1016.599,179.252,-124.941,167.454,53.323,159.901
C09506=1016.604,179.501,-124.962,167.458,53.313,159.900
C09507=1016.609,179.750,-124.984,167.462,53.304,159.899
C09508=1016.614,179.999,-125.004,167.466,53.294,159.897
C09509=1016.619,180.248,-125.026,167.470,53.284,159.896
C09510=1016.624,180.497,-125.047,167.475,53.273,159.895
C09511=1016.629,180.746,-125.068,167.478,53.263,159.894
C09512=1016.633,180.995,-125.089,167.482,53.253,159.892
C09513=1016.638,181.244,-125.111,167.487,53.244,159.891
C09514=1016.643,181.493,-125.132,167.491,53.234,159.890
C09515=1016.648,181.742,-125.153,167.495,53.223,159.889
C09516=1016.653,181.992,-125.175,167.499,53.213,159.888
C09517=1016.658,182.240,-125.196,167.503,53.204,159.887
C09518=1016.661,182.490,-125.218,167.507,53.194,159.885
C09519=1016.666,182.738,-125.240,167.512,53.184,159.884
C09520=1016.670,182.987,-125.262,167.516,53.174,159.883
C09521=1016.674,183.237,-125.283,167.520,53.165,159.882
C09522=1016.679,183.486,-125.305,167.523,53.155,159.881
C09523=1016.684,183.735,-125.327,167.529,53.145,159.880
C09524=1016.689,183.983,-125.349,167.532,53.135,159.879
C09525=1016.693,184.232,-125.371,167.536,53.126,159.878
C09526=1016.697,184.482,-125.393,167.540,53.116,159.876
C09527=1016.702,184.731,-125.414,167.545,53.106,159.875
C09528=1016.707,184.980,-125.436,167.549,53.097,159.874
C09529=1016.711,185.229,-125.459,167.553,53.087,159.873
C09530=1016.716,185.477,-125.481,167.557,53.077,159.872
C09531=1016.720,185.727,-125.502,167.561,53.067,159.871
C09532=1016.724,185.976,-125.524,167.566,53.058,159.869
C09533=1016.729,186.225,-125.546,167.569,53.048,159.868
C09534=1016.734,186.474,-125.568,167.574,53.038,159.867
C09535=1016.739,186.754,-125.592,167.579,53.027,159.866
C09536=1016.744,187.034,-125.618,167.583,53.016,159.865
C09537=1016.750,187.315,-125.642,167.589,53.005,159.863
C09538=1016.754,187.594,-125.667,167.593,52.994,159.862
C09539=1016.759,187.844,-125.688,167.597,52.984,159.861
C09540=1016.764,188.093,-125.710,167.602,52.975,159.860
C09541=1016.768,188.341,-125.732,167.606,52.965,159.859
C09542=1016.772,188.590,-125.754,167.610,52.956,159.858
C09543=1016.778,188.840,-125.777,167.614,52.945,159.856
C09544=1016.783,189.089,-125.799,167.619,52.936,159.855
C09545=1016.787,189.338,-125.820,167.623,52.926,159.854
C09546=1016.792,189.587,-125.843,167.628,52.916,159.853
C09547=1016.796,189.836,-125.865,167.631,52.907,159.852
C09548=1016.801,190.084,-125.887,167.636,52.897,159.851
C09549=1016.805,190.333,-125.909,167.640,52.887,159.850
C09550=1016.810,190.582,-125.931,167.644,52.878,159.849
C09551=1016.815,190.831,-125.953,167.649,52.867,159.847
C09552=1016.820,191.080,-125.975,167.653,52.858,159.846
C09553=1016.824,191.330,-125.997,167.658,52.848,159.845
C09554=1016.829,191.579,-126.019,167.662,52.839,159.844
C09555=1016.834,191.827,-126.041,167.666,52.829,159.843
C09556=1016.838,192.077,-126.064,167.671,52.819,159.842
C09557=1016.843,192.325,-126.086,167.675,52.809,159.841
C09558=1016.848,192.574,-126.107,167.680,52.799,159.840
C09559=1016.854,192.823,-126.130,167.684,52.790,159.838
C09560=1016.858,193.072,-126.153,167.689,52.780,159.837
C09561=1016.862,193.321,-126.175,167.693,52.770,159.836
C09562=1016.867,193.570,-126.197,167.698,52.760,159.835
C09563=1016.871,193.819,-126.219,167.702,52.751,159.834
C09564=1016.877,194.068,-126.241,167.706,52.741,159.833
C09565=1016.882,194.317,-126.263,167.711,52.731,159.832
C09566=1016.886,194.566,-126.286,167.715,52.722,159.831
C09567=1016.891,194.815,-126.308,167.720,52.712,159.830
C09568=1016.896,195.063,-126.330,167.724,52.702,159.828
C09569=1016.901,195.313,-126.352,167.729,52.693,159.827
C09570=1016.905,195.562,-126.375,167.733,52.683,159.826
C09571=1016.910,195.811,-126.397,167.738,52.673,159.825
C09572=1016.915,196.059,-126.419,167.742,52.663,159.824
C09573=1016.920,196.309,-126.442,167.747,52.654,159.823
C09574=1016.925,196.558,-126.464,167.751,52.644,159.822
C09575=1016.929,196.806,-126.486,167.756,52.634,159.821
C09576=1016.934,197.056,-126.509,167.760,52.624,159.819
C09577=1016.939,197.305,-126.531,167.765,52.615,159.819
C09578=1016.944,197.553,-126.553,167.769,52.605,159.817
C09579=1016.950,197.802,-126.576,167.774,52.595,159.816
C09580=1016.954,198.051,-126.598,167.779,52.585,159.815
C09581=1016.959,198.300,-126.620,167.783,52.576,159.814
C09582=1016.964,198.549,-126.643,167.788,52.566,159.813
C09583=1016.969,198.798,-126.666,167.792,52.556,159.812
C09584=1016.973,199.047,-126.687,167.797,52.546,159.811
C09585=1016.979,199.296,-126.710,167.801,52.537,159.810
C09586=1016.983,199.545,-126.733,167.806,52.527,159.809
C09587=1016.988,199.794,-126.756,167.810,52.518,159.808
C09588=1016.992,200.043,-126.779,167.816,52.508,159.807
C09589=1016.997,200.292,-126.801,167.819,52.499,159.805
C09590=1017.002,200.541,-126.824,167.825,52.489,159.804
C09591=1017.006,200.790,-126.847,167.829,52.480,159.803
C09592=1017.012,201.038,-126.870,167.834,52.470,159.802
C09593=1017.016,201.287,-126.892,167.838,52.460,159.801
C09594=1017.021,201.536,-126.916,167.843,52.451,159.800
C09595=1017.026,201.785,-126.939,167.847,52.441,159.799
C09596=1017.030,202.033,-126.962,167.852,52.432,159.798
C09597=1017.035,202.281,-126.984,167.857,52.423,159.797
C09598=1017.058,203.524,-127.098,168.348,52.501,159.911
C09599=1017.064,203.761,-127.122,168.352,52.493,159.910
C09600=1017.070,203.999,-127.145,168.356,52.485,159.909
C09601=1017.075,204.236,-127.168,168.359,52.477,159.908
C09602=1017.081,204.474,-127.192,168.364,52.469,159.907
C09603=1017.086,204.712,-127.215,168.368,52.461,159.906
C09604=1017.092,204.949,-127.239,168.371,52.453,159.905
C09605=1017.097,205.187,-127.263,168.375,52.445,159.904
C09606=1017.103,205.425,-127.286,168.379,52.437,159.903
C09607=1017.109,205.673,-127.311,168.383,52.429,159.902
C09608=1017.114,205.922,-127.335,168.387,52.421,159.901
C09609=1017.120,206.171,-127.360,168.390,52.413,159.900
C09610=1017.126,206.419,-127.385,168.395,52.404,159.899
C09611=1017.132,206.668,-127.410,168.399,52.396,159.898
C09612=1017.138,206.916,-127.434,168.403,52.387,159.897
C09613=1017.144,207.165,-127.459,168.407,52.379,159.896
C09614=1017.149,207.413,-127.484,168.411,52.371,159.895
C09615=1017.155,207.663,-127.509,168.415,52.362,159.894
C09616=1017.160,207.912,-127.533,168.418,52.354,159.893
C09617=1017.166,208.160,-127.558,168.423,52.346,159.892
C09618=1017.172,208.409,-127.583,168.427,52.338,159.891
C09619=1017.178,208.657,-127.608,168.431,52.330,159.890
C09620=1017.183,208.907,-127.633,168.435,52.322,159.889
C09621=1017.189,209.155,-127.658,168.439,52.314,159.888
C09622=1017.195,209.404,-127.682,168.444,52.306,159.888
C09623=1017.201,209.653,-127.708,168.447,52.298,159.887
C09624=1017.207,209.901,-127.732,168.451,52.290,159.886
C09625=1017.212,210.150,-127.758,168.456,52.281,159.885
C09626=1017.218,210.398,-127.783,168.459,52.273,159.884
C09627=1017.224,210.647,-127.808,168.463,52.265,159.883
C09628=1017.230,210.896,-127.833,168.468,52.258,159.882
C09629=1017.235,211.144,-127.858,168.472,52.250,159.881
C09630=1017.241,211.393,-127.884,168.475,52.242,159.880
C09631=1017.246,211.642,-127.908,168.479,52.234,159.879
C09632=1017.252,211.890,-127.933,168.484,52.226,159.878
C09633=1017.258,212.139,-127.959,168.488,52.218,159.877
C09634=1017.263,212.388,-127.983,168.491,52.210,159.876
C09635=1017.269,212.636,-128.009,168.496,52.202,159.875
C09636=1017.275,212.885,-128.034,168.500,52.194,159.875
C09637=1017.280,213.133,-128.060,168.504,52.186,159.874
C09638=1017.286,213.383,-128.084,168.507,52.178,159.873
C09639=1017.292,213.631,-128.110,168.513,52.171,159.872
C09640=1017.298,213.879,-128.134,168.516,52.163,159.871
C09641=1017.303,214.128,-128.160,168.520,52.155,159.870
C09642=1017.310,214.377,-128.186,168.524,52.147,159.869
C09643=1017.316,214.626,-128.210,168.529,52.139,159.868
C09644=1017.321,214.874,-128.235,168.533,52.132,159.867
C09645=1017.327,215.123,-128.261,168.536,52.124,159.866
C09646=1017.333,215.372,-128.287,168.540,52.116,159.865
C09647=1017.338,215.620,-128.312,168.545,52.108,159.865
C09648=1017.345,215.869,-128.337,168.549,52.100,159.864
C09649=1017.350,216.118,-128.362,168.553,52.093,159.863
C09650=1017.356,216.367,-128.387,168.557,52.085,159.862
C09651=1017.362,216.615,-128.412,168.562,52.077,159.861
C09652=1017.367,216.864,-128.438,168.565,52.069,159.860
C09653=1017.373,217.112,-128.464,168.570,52.062,159.859
C09654=1017.379,217.361,-128.489,168.573,52.054,159.858
C09655=1017.385,217.609,-128.514,168.578,52.046,159.858
C09656=1017.391,217.858,-128.540,168.582,52.038,159.857
C09657=1017.397,218.107,-128.565,168.586,52.031,159.856
C09658=1017.403,218.355,-128.591,168.590,52.023,159.855
C09659=1017.408,218.590,-128.615,168.594,52.016,159.854
C09660=1017.414,218.824,-128.639,168.598,52.008,159.853
C09661=1017.419,219.059,-128.663,168.602,52.002,159.853
C09662=1017.424,219.294,-128.687,168.606,51.995,159.852
C09663=1017.429,219.528,-128.712,168.610,51.987,159.851
C09664=1017.434,219.763,-128.737,168.613,51.980,159.850
C09665=1017.440,219.998,-128.760,168.617,51.973,159.849
C09666=1017.445,220.233,-128.785,168.621,51.966,159.849
C09667=1017.451,220.481,-128.810,168.625,51.959,159.848
C09668=1017.457,220.729,-128.837,168.629,51.951,159.847
C09669=1017.463,220.978,-128.862,168.634,51.944,159.846
C09670=1017.469,221.227,-128.888,168.637,51.936,159.845
C09671=1017.475,221.476,-128.913,168.641,51.929,159.844
C09672=1017.480,221.724,-128.939,168.647,51.921,159.844
C09673=1017.487,221.973,-128.965,168.651,51.914,159.843
C09674=1017.492,222.221,-128.991,168.655,51.907,159.842
C09675=1017.497,222.470,-129.017,168.659,51.899,159.841
C09676=1017.503,222.718,-129.042,168.663,51.891,159.840
C09677=1017.509,222.967,-129.069,168.667,51.884,159.840
C09678=1017.515,223.215,-129.094,168.671,51.877,159.839
C09679=1017.521,223.464,-129.120,168.675,51.870,159.838
C09680=1017.527,223.713,-129.145,168.679,51.862,159.837
C09681=1017.533,223.961,-129.172,168.683,51.855,159.836
C09682=1017.538,224.210,-129.198,168.687,51.848,159.836
C09683=1017.544,224.459,-129.223,168.692,51.841,159.835
C09684=1017.550,224.708,-129.250,168.697,51.833,159.834
C09685=1017.556,224.956,-129.275,168.701,51.826,159.833
C09686=1017.561,225.204,-129.301,168.705,51.818,159.833
C09687=1017.567,225.453,-129.327,168.709,51.811,159.831
C09688=1017.573,225.701,-129.353,168.713,51.803,159.831
C09689=1017.579,225.950,-129.379,168.717,51.796,159.830
C09690=1017.585,226.199,-129.405,168.721,51.789,159.829
C09691=1017.591,226.447,-129.431,168.725,51.782,159.828
C09692=1017.596,226.696,-129.457,168.730,51.775,159.828
C09693=1017.603,226.944,-129.483,168.734,51.768,159.827
C09694=1017.608,227.193,-129.509,168.738,51.760,159.826
C09695=1017.614,227.441,-129.536,168.742,51.753,159.825
C09696=1017.620,227.690,-129.562,168.747,51.746,159.825
C09697=1017.625,227.939,-129.589,168.751,51.739,159.824
C09698=1017.631,228.188,-129.614,168.755,51.732,159.823
C09699=1017.637,228.436,-129.641,168.759,51.725,159.822
C09700=1017.643,228.684,-129.667,168.764,51.718,159.822
C09701=1017.649,228.933,-129.693,168.768,51.710,159.821
C09702=1017.654,229.181,-129.720,168.772,51.704,159.820
C09703=1017.660,229.430,-129.746,168.776,51.697,159.819
C09704=1017.666,229.679,-129.772,168.781,51.689,159.819
C09705=1017.672,229.927,-129.798,168.785,51.682,159.818
C09706=1017.678,230.175,-129.825,168.788,51.676,159.817
C09707=1017.683,230.424,-129.851,168.793,51.669,159.816
C09708=1017.690,230.673,-129.878,168.797,51.662,159.816
C09709=1017.696,230.921,-129.905,168.801,51.655,159.815
C09710=1017.701,231.170,-129.931,168.805,51.648,159.814
C09711=1017.707,231.419,-129.957,168.810,51.641,159.814
C09712=1017.713,231.667,-129.984,168.814,51.634,159.813
C09713=1017.718,231.916,-130.010,168.818,51.627,159.812
C09714=1017.724,232.164,-130.037,168.823,51.620,159.812
C09715=1017.730,232.412,-130.064,168.827,51.613,159.811
C09716=1017.736,232.661,-130.090,168.832,51.606,159.810
C09717=1017.741,232.910,-130.116,168.835,51.600,159.809
C09718=1017.747,233.159,-130.143,168.840,51.593,159.809
C09719=1017.752,233.389,-130.168,168.844,51.586,159.808
C09720=1017.758,233.619,-130.193,168.848,51.580,159.807
C09721=1017.764,233.850,-130.217,168.851,51.574,159.807
C09722=1017.769,234.080,-130.242,168.856,51.568,159.806
C09723=1017.774,234.310,-130.267,168.859,51.561,159.805
C09724=1017.780,234.542,-130.291,168.864,51.555,159.805
C09725=1017.785,234.772,-130.316,168.868,51.549,159.804
C09726=1017.790,235.002,-130.341,168.871,51.543,159.804
C09727=1017.797,235.251,-130.368,168.875,51.535,159.803
C09728=1017.802,235.499,-130.395,168.880,51.529,159.802
C09729=1017.808,235.748,-130.421,168.884,51.522,159.801
C09730=1017.814,235.996,-130.448,168.889,51.515,159.801
C09731=1017.820,236.244,-130.475,168.893,51.509,159.800
C09732=1017.826,236.493,-130.502,168.898,51.501,159.799
C09733=1017.832,236.742,-130.528,168.901,51.495,159.799
C09734=1017.838,236.990,-130.555,168.906,51.489,159.798
C09735=1017.843,237.238,-130.582,168.910,51.481,159.797
C09736=1017.850,237.488,-130.609,168.915,51.475,159.797
C09737=1017.856,237.736,-130.635,168.919,51.468,159.796
C09738=1017.861,237.984,-130.662,168.923,51.461,159.795
C09739=1017.867,238.232,-130.689,168.928,51.455,159.795
C09740=1017.873,238.480,-130.716,168.932,51.449,159.794
C09741=1017.880,238.729,-130.743,168.936,51.442,159.794
C09742=1017.885,238.978,-130.770,168.940,51.435,159.793
C09743=1017.890,239.226,-130.797,168.945,51.428,159.792
C09744=1017.896,239.474,-130.824,168.950,51.422,159.792
C09745=1017.903,239.723,-130.851,168.953,51.416,159.791
C09746=1017.908,239.972,-130.879,168.958,51.409,159.790
C09747=1017.914,240.220,-130.906,168.963,51.403,159.790
C09748=1017.920,240.469,-130.933,168.967,51.396,159.789
C09749=1017.925,240.717,-130.960,168.971,51.390,159.788
C09750=1017.931,240.965,-130.987,168.975,51.383,159.788
C09751=1017.937,241.213,-131.014,168.980,51.377,159.787
C09752=1017.943,241.463,-131.042,168.985,51.370,159.787
C09753=1017.949,241.711,-131.069,168.988,51.364,159.786
C09754=1017.955,241.959,-131.096,168.993,51.358,159.785
C09755=1017.961,242.208,-131.124,168.997,51.351,159.785
C09756=1017.966,242.456,-131.151,169.002,51.345,159.784
C09757=1017.972,242.704,-131.177,169.006,51.339,159.784
C09758=1017.978,242.953,-131.206,169.010,51.332,159.783
C09759=1017.984,243.202,-131.232,169.015,51.326,159.782
C09760=1017.989,243.450,-131.260,169.020,51.319,159.782
C09761=1017.996,243.699,-131.287,169.023,51.313,159.781
C09762=1018.001,243.947,-131.315,169.028,51.307,159.781
C09763=1018.007,244.195,-131.344,169.033,51.301,159.780
C09764=1018.013,244.444,-131.370,169.036,51.295,159.780
C09765=1018.018,244.692,-131.398,169.041,51.288,159.779
C09766=1018.025,244.940,-131.426,169.046,51.282,159.778
C09767=1018.030,245.189,-131.453,169.050,51.276,159.778
C09768=1018.035,245.437,-131.481,169.054,51.270,159.777
C09769=1018.042,245.685,-131.509,169.059,51.263,159.777
C09770=1018.047,245.934,-131.536,169.063,51.257,159.776
C09771=1018.053,246.183,-131.564,169.068,51.251,159.776
C09772=1018.059,246.431,-131.592,169.072,51.245,159.775
C09773=1018.064,246.680,-131.619,169.076,51.239,159.774
C09774=1018.070,246.928,-131.647,169.081,51.233,159.774
C09775=1018.076,247.176,-131.675,169.086,51.226,159.773
C09776=1018.082,247.425,-131.703,169.089,51.220,159.773
C09777=1018.088,247.672,-131.730,169.094,51.214,159.772
C09778=1018.093,247.922,-131.758,169.099,51.208,159.772
C09779=1018.099,248.148,-131.784,169.103,51.203,159.771
C09780=1018.104,248.376,-131.809,169.107,51.197,159.771
C09781=1018.110,248.603,-131.835,169.111,51.192,159.770
C09782=1018.115,248.830,-131.859,169.115,51.186,159.770
C09783=1018.121,249.057,-131.885,169.119,51.181,159.769
C09784=1018.126,249.284,-131.910,169.123,51.175,159.769
C09785=1018.131,249.511,-131.936,169.127,51.169,159.768
C09786=1018.137,249.739,-131.962,169.131,51.164,159.768
C09787=1018.142,249.987,-131.990,169.136,51.158,159.767
C09788=1018.149,250.236,-132.017,169.141,51.151,159.767
C09789=1018.154,250.484,-132.045,169.145,51.146,159.766
C09790=1018.160,250.733,-132.073,169.149,51.140,159.766
C09791=1018.166,250.980,-132.101,169.153,51.134,159.765
C09792=1018.172,251.229,-132.129,169.158,51.128,159.765
C09793=1018.179,251.478,-132.157,169.163,51.122,159.764
C09794=1018.184,251.726,-132.185,169.167,51.116,159.764
C09795=1018.190,251.974,-132.213,169.172,51.110,159.763
C09796=1018.196,252.222,-132.240,169.176,51.104,159.763
C09797=1018.202,252.471,-132.269,169.180,51.098,159.762
C09798=1018.208,252.720,-132.297,169.185,51.092,159.762
C09799=1018.214,252.967,-132.324,169.190,51.086,159.761
C09800=1018.220,253.216,-132.353,169.194,51.080,159.761
C09801=1018.226,253.465,-132.381,169.199,51.074,159.760
C09802=1018.232,253.713,-132.408,169.204,51.068,159.760
C09803=1018.238,253.961,-132.437,169.208,51.063,159.759
C09804=1018.244,254.210,-132.464,169.213,51.056,159.759
C09805=1018.250,254.458,-132.492,169.217,51.051,159.758
C09806=1018.256,254.707,-132.521,169.222,51.045,159.758
C09807=1018.263,254.954,-132.549,169.226,51.039,159.757
C09808=1018.268,255.202,-132.577,169.230,51.033,159.757
C09809=1018.274,255.451,-132.605,169.235,51.027,159.756
C09810=1018.281,255.700,-132.633,169.240,51.021,159.756
C09811=1018.286,255.948,-132.661,169.244,51.016,159.755
C09812=1018.292,256.196,-132.689,169.249,51.010,159.755
C09813=1018.299,256.445,-132.717,169.254,51.004,159.755
C09814=1018.305,256.693,-132.746,169.258,50.998,159.754
C09815=1018.310,256.941,-132.774,169.263,50.992,159.754
C09816=1018.317,257.190,-132.802,169.267,50.987,159.753
C09817=1018.323,257.438,-132.830,169.272,50.981,159.753
C09818=1018.329,257.686,-132.859,169.277,50.975,159.752
C09819=1018.335,257.934,-132.887,169.281,50.969,159.752
C09820=1018.341,258.183,-132.915,169.286,50.963,159.751
C09821=1018.348,258.431,-132.943,169.291,50.958,159.751
C09822=1018.354,258.679,-132.972,169.295,50.952,159.750
C09823=1018.360,258.928,-133.000,169.300,50.946,159.750
C09824=1018.366,259.176,-133.027,169.304,50.940,159.749
C09825=1018.372,259.424,-133.056,169.309,50.935,159.749
C09826=1018.378,259.673,-133.085,169.314,50.929,159.749
C09827=1018.385,259.921,-133.112,169.318,50.923,159.748
C09828=1018.391,260.169,-133.141,169.323,50.918,159.748
C09829=1018.396,260.418,-133.170,169.327,50.912,159.747
C09830=1018.402,260.666,-133.199,169.332,50.907,159.747
C09831=1018.408,260.914,-133.228,169.337,50.902,159.747
C09832=1018.414,261.163,-133.256,169.342,50.896,159.746
C09833=1018.420,261.411,-133.285,169.346,50.891,159.746
C09834=1018.426,261.660,-133.314,169.351,50.885,159.745
C09835=1018.432,261.907,-133.342,169.356,50.879,159.745
C09836=1018.438,262.155,-133.372,169.360,50.874,159.744
C09837=1018.444,262.404,-133.400,169.365,50.868,159.744
C09838=1018.451,262.652,-133.429,169.370,50.863,159.744
C09839=1018.459,262.988,-133.468,169.376,50.856,159.743
C09840=1018.467,263.323,-133.507,169.383,50.848,159.743
C09841=1018.475,263.658,-133.546,169.389,50.841,159.742
C09842=1018.484,263.994,-133.585,169.395,50.834,159.742
C09843=1018.490,264.243,-133.613,169.400,50.828,159.741
C09844=1018.495,264.491,-133.643,169.404,50.823,159.741
C09845=1018.501,264.739,-133.672,169.409,50.818,159.741
C09846=1018.508,264.987,-133.701,169.413,50.812,159.740
C09847=1018.514,265.236,-133.729,169.418,50.807,159.740
C09848=1018.519,265.483,-133.758,169.424,50.802,159.740
C09849=1018.525,265.732,-133.787,169.428,50.796,159.739
C09850=1018.532,265.980,-133.816,169.432,50.791,159.739
C09851=1018.537,266.228,-133.846,169.438,50.786,159.738
C09852=1018.543,266.476,-133.875,169.442,50.780,159.738
C09853=1018.550,266.724,-133.904,169.447,50.775,159.738
C09854=1018.556,266.973,-133.933,169.451,50.770,159.737
C09855=1018.561,267.221,-133.962,169.457,50.765,159.737
C09856=1018.568,267.469,-133.992,169.461,50.759,159.737
C09857=1018.574,267.717,-134.021,169.466,50.754,159.736
C09858=1018.580,267.965,-134.050,169.470,50.749,159.736
C09859=1018.586,268.214,-134.079,169.476,50.744,159.736
C09860=1018.592,268.462,-134.108,169.480,50.739,159.735
C09861=1018.598,268.710,-134.137,169.485,50.733,159.735
C09862=1018.604,268.958,-134.166,169.489,50.728,159.735
C09863=1018.613,269.325,-134.210,169.497,50.721,159.734
C09864=1018.623,269.689,-134.253,169.503,50.713,159.734
C09865=1018.631,270.055,-134.296,169.511,50.706,159.733
C09866=1018.640,270.419,-134.340,169.518,50.698,159.733
C09867=1018.646,270.668,-134.369,169.523,50.693,159.732
C09868=1018.652,270.916,-134.398,169.528,50.688,159.732
C09869=1018.659,271.164,-134.428,169.533,50.682,159.732
C09870=1018.665,271.413,-134.458,169.537,50.678,159.732
C09871=1018.671,271.661,-134.487,169.543,50.673,159.731
C09872=1018.676,271.909,-134.517,169.547,50.668,159.731
C09873=1018.683,272.157,-134.546,169.552,50.662,159.731
C09874=1018.688,272.405,-134.576,169.557,50.657,159.730
C09875=1018.695,272.653,-134.605,169.561,50.653,159.730
C09876=1018.701,272.901,-134.635,169.567,50.648,159.730
C09877=1018.707,273.149,-134.665,169.571,50.643,159.730
C09878=1018.713,273.398,-134.695,169.576,50.637,159.729
C09879=1018.719,273.646,-134.724,169.581,50.633,159.729
C09880=1018.725,273.894,-134.754,169.586,50.628,159.729
C09881=1018.732,274.142,-134.784,169.591,50.623,159.729
C09882=1018.737,274.390,-134.813,169.596,50.618,159.728
C09883=1018.744,274.639,-134.843,169.601,50.613,159.728
C09884=1018.750,274.887,-134.873,169.605,50.608,159.728
C09885=1018.756,275.135,-134.903,169.611,50.603,159.728
C09886=1018.762,275.383,-134.932,169.615,50.599,159.727
C09887=1018.768,275.630,-134.962,169.621,50.594,159.727
C09888=1018.774,275.880,-134.992,169.625,50.589,159.727
C09889=1018.781,276.127,-135.022,169.631,50.584,159.727
C09890=1018.786,276.376,-135.052,169.635,50.579,159.726
C09891=1018.793,276.623,-135.081,169.641,50.574,159.726
C09892=1018.799,276.872,-135.112,169.645,50.570,159.726
C09893=1018.805,277.119,-135.142,169.650,50.565,159.726
C09894=1018.812,277.368,-135.171,169.655,50.560,159.725
C09895=1018.817,277.596,-135.199,169.659,50.555,159.725
C09896=1018.823,277.825,-135.228,169.664,50.551,159.725
C09897=1018.828,278.053,-135.255,169.668,50.547,159.725
C09898=1018.834,278.282,-135.283,169.673,50.543,159.725
C09899=1018.839,278.510,-135.311,169.677,50.538,159.724
C09900=1018.845,278.740,-135.339,169.682,50.534,159.724
C09901=1018.851,278.968,-135.366,169.687,50.529,159.724
C09902=1018.856,279.196,-135.395,169.691,50.525,159.724
C09903=1018.862,279.445,-135.425,169.696,50.521,159.724
C09904=1018.869,279.693,-135.454,169.701,50.516,159.723
C09905=1018.875,279.941,-135.485,169.706,50.511,159.723
C09906=1018.881,280.189,-135.515,169.712,50.507,159.723
C09907=1018.887,280.437,-135.546,169.716,50.502,159.723
C09908=1018.894,280.684,-135.575,169.721,50.497,159.723
C09909=1018.900,280.933,-135.606,169.726,50.492,159.722
C09910=1018.906,281.181,-135.637,169.731,50.488,159.722
C09911=1018.912,281.429,-135.667,169.737,50.483,159.722
C09912=1018.919,281.677,-135.697,169.741,50.478,159.722
C09913=1018.925,281.925,-135.727,169.746,50.474,159.722
C09914=1018.931,282.173,-135.758,169.752,50.469,159.722
C09915=1018.937,282.421,-135.788,169.756,50.465,159.721
C09916=1018.944,282.669,-135.819,169.762,50.460,159.721
C09917=1018.950,282.917,-135.849,169.766,50.456,159.721
C09918=1018.956,283.165,-135.880,169.771,50.452,159.721
C09919=1018.962,283.413,-135.910,169.777,50.447,159.721
C09920=1018.968,283.662,-135.941,169.781,50.442,159.720
C09921=1018.975,283.909,-135.970,169.787,50.438,159.720
C09922=1018.981,284.158,-136.001,169.792,50.433,159.720
C09923=1018.987,284.406,-136.032,169.798,50.429,159.720
C09924=1018.994,284.654,-136.062,169.802,50.424,159.720
C09925=1019.000,284.902,-136.092,169.807,50.420,159.720
C09926=1019.007,285.150,-136.123,169.813,50.415,159.720
C09927=1019.013,285.397,-136.154,169.817,50.411,159.720
C09928=1019.019,285.646,-136.185,169.822,50.407,159.719
C09929=1019.025,285.893,-136.216,169.828,50.402,159.719
C09930=1019.032,286.142,-136.246,169.833,50.398,159.719
C09931=1019.037,286.390,-136.277,169.838,50.393,159.719
C09932=1019.044,286.637,-136.308,169.843,50.389,159.719
C09933=1019.050,286.885,-136.338,169.848,50.385,159.719
C09934=1019.056,287.134,-136.369,169.853,50.380,159.719
C09935=1019.063,287.381,-136.400,169.858,50.376,159.719
C09936=1019.069,287.629,-136.431,169.864,50.372,159.719
C09937=1019.076,287.877,-136.462,169.869,50.368,159.718
C09938=1019.081,288.126,-136.493,169.874,50.363,159.718
C09939=1019.087,288.374,-136.524,169.880,50.359,159.718
C09940=1019.093,288.621,-136.555,169.884,50.355,159.718
C09941=1019.100,288.870,-136.586,169.889,50.351,159.718
C09942=1019.106,289.118,-136.617,169.895,50.346,159.718
C09943=1019.112,289.365,-136.648,169.900,50.342,159.718
C09944=1019.119,289.613,-136.679,169.906,50.337,159.718
C09945=1019.126,289.861,-136.710,169.910,50.333,159.718
C09946=1019.132,290.109,-136.741,169.915,50.329,159.718
C09947=1019.138,290.357,-136.772,169.921,50.325,159.718
C09948=1019.145,290.606,-136.803,169.926,50.320,159.717
C09949=1019.151,290.853,-136.834,169.932,50.316,159.717
C09950=1019.157,291.101,-136.866,169.937,50.312,159.717
C09951=1019.163,291.349,-136.897,169.941,50.308,159.717
C09952=1019.169,291.597,-136.928,169.947,50.304,159.717
C09953=1019.176,291.845,-136.959,169.952,50.300,159.717
C09954=1019.182,292.093,-136.990,169.957,50.296,159.717
C09955=1019.188,292.328,-137.020,169.962,50.292,159.717
C09956=1019.194,292.562,-137.050,169.968,50.288,159.717
C09957=1019.200,292.796,-137.079,169.973,50.284,159.717
C09958=1019.207,293.031,-137.109,169.978,50.280,159.717
C09959=1019.212,293.266,-137.139,169.983,50.276,159.717
C09960=1019.218,293.501,-137.169,169.988,50.273,159.717
C09961=1019.224,293.736,-137.199,169.993,50.269,159.717
C09962=1019.229,293.971,-137.229,169.998,50.265,159.717
C09963=1019.236,294.219,-137.260,170.003,50.261,159.717
C09964=1019.242,294.467,-137.292,170.008,50.257,159.717
C09965=1019.248,294.714,-137.324,170.013,50.253,159.717
C09966=1019.254,294.962,-137.355,170.019,50.249,159.717
C09967=1019.261,295.210,-137.388,170.024,50.246,159.717
C09968=1019.267,295.458,-137.419,170.029,50.242,159.717
C09969=1019.273,295.705,-137.451,170.035,50.237,159.717
C09970=1019.279,295.953,-137.482,170.040,50.233,159.717
C09971=1019.285,296.201,-137.514,170.045,50.230,159.717
C09972=1019.292,296.449,-137.546,170.051,50.226,159.717
C09973=1019.298,296.697,-137.578,170.056,50.222,159.717
C09974=1019.304,296.945,-137.611,170.061,50.218,159.717
C09975=1019.311,297.192,-137.642,170.067,50.214,159.717
C09976=1019.317,297.440,-137.674,170.072,50.211,159.717
C09977=1019.323,297.688,-137.705,170.077,50.207,159.717
C09978=1019.330,297.936,-137.738,170.083,50.202,159.717
C09979=1019.336,298.184,-137.769,170.088,50.199,159.717
C09980=1019.342,298.432,-137.801,170.093,50.195,159.717
C09981=1019.348,298.680,-137.833,170.100,50.191,159.717
C09982=1019.355,298.928,-137.866,170.105,50.187,159.717
C09983=1019.361,299.176,-137.898,170.111,50.184,159.717
C09984=1019.368,299.424,-137.929,170.116,50.180,159.717
C09985=1019.374,299.671,-137.962,170.121,50.176,159.717
C09986=1019.381,299.919,-137.993,170.127,50.172,159.717
C09987=1019.387,300.167,-138.026,170.132,50.169,159.717
C09988=1019.393,300.414,-138.058,170.137,50.165,159.717
C09989=1019.399,300.662,-138.089,170.143,50.161,159.717
C09990=1019.406,300.910,-138.122,170.148,50.157,159.717
C09991=1019.413,301.158,-138.154,170.154,50.154,159.717
C09992=1019.419,301.406,-138.186,170.160,50.150,159.718
C09993=1019.426,301.654,-138.218,170.165,50.146,159.717
C09994=1019.432,301.901,-138.250,170.171,50.143,159.718
C09995=1019.438,302.150,-138.282,170.176,50.139,159.718
C09996=1019.445,302.397,-138.315,170.181,50.135,159.718
//INST
///DATE 2021/06/17 10:59
///ATTR SC,RW,RJ
////FRAME ROBOT
///GROUP1 RB1
NOP
MOVL C00000 V=800.0 PL=0
MOVL C00001 V=800.0 PL=0
MOVL C00002 V=800.0 PL=0
MOVL C00003 V=800.0 PL=0
MOVL C00004 V=800.0 PL=0
MOVL C00005 V=800.0 PL=0
MOVL C00006 V=800.0 PL=0
MOVL C00007 V=800.0 PL=0
MOVL C00008 V=800.0 PL=0
MOVL C00009 V=800.0 PL=0
MOVL C00010 V=800.0 PL=0
MOVL C00011 V=800.0 PL=0
MOVL C00012 V=800.0 PL=0
MOVL C00013 V=800.0 PL=0
MOVL C00014 V=800.0 PL=0
MOVL C00015 V=800.0 PL=0
MOVL C00016 V=800.0 PL=0
MOVL C00017 V=800.0 PL=0
MOVL C00018 V=800.0 PL=0
MOVL C00019 V=800.0 PL=0
MOVL C00020 V=800.0 PL=0
MOVL C00021 V=800.0 PL=0
MOVL C00022 V=800.0 PL=0
MOVL C00023 V=800.0 PL=0
MOVL C00024 V=800.0 PL=0
MOVL C00025 V=800.0 PL=0
MOVL C00026 V=800.0 PL=0
MOVL C00027 V=800.0 PL=0
MOVL C00028 V=800.0 PL=0
MOVL C00029 V=800.0 PL=0
MOVL C00030 V=800.0 PL=0
MOVL C00031 V=800.0 PL=0
MOVL C00032 V=800.0 PL=0
MOVL C00033 V=800.0 PL=0
MOVL C00034 V=800.0 PL=0
MOVL C00035 V=800.0 PL=0
MOVL C00036 V=800.0 PL=0
MOVL C00037 V=800.0 PL=0
MOVL C00038 V=800.0 PL=0
MOVL C00039 V=800.0 PL=0
MOVL C00040 V=800.0 PL=0
MOVL C00041 V=800.0 PL=0
MOVL C00042 V=800.0 PL=0
MOVL C00043 V=800.0 PL=0
MOVL C00044 V=800.0 PL=0
MOVL C00045 V=800.0 PL=0
MOVL C00046 V=800.0 PL=0
MOVL C00047 V=800.0 PL=0
MOVL C00048 V=800.0 PL=0
MOVL C00049 V=800.0 PL=0
MOVL C00050 V=800.0 PL=0
MOVL C00051 V=800.0 PL=0
MOVL C00052 V=800.0 PL=0
MOVL C00053 V=800.0 PL=0
MOVL C00054 V=800.0 PL=0
MOVL C00055 V=800.0 PL=0
MOVL C00056 V=800.0 PL=0
MOVL C00057 V=800.0 PL=0
MOVL C00058 V=800.0 PL=0
MOVL C00059 V=800.0 PL=0
MOVL C00060 V=800.0 PL=0
MOVL C00061 V=800.0 PL=0
MOVL C00062 V=800.0 PL=0
MOVL C00063 V=800.0 PL=0
MOVL C00064 V=800.0 PL=0
MOVL C00065 V=800.0 PL=0
MOVL C00066 V=800.0 PL=0
MOVL C00067 V=800.0 PL=0
MOVL C00068 V=800.0 PL=0
MOVL C00069 V=800.0 PL=0
MOVL C00070 V=800.0 PL=0
MOVL C00071 V=800.0 PL=0
MOVL C00072 V=800.0 PL=0
MOVL C00073 V=800.0 PL=0
MOVL C00074 V=800.0 PL=0
MOVL C00075 V=800.0 PL=0
MOVL C00076 V=800.0 PL=0
MOVL C00077 V=800.0 PL=0
MOVL C00078 V=800.0 PL=0
MOVL C00079 V=800.0 PL=0
MOVL C00080 V=800.0 PL=0
MOVL C00081 V=800.0 PL=0
MOVL C00082 V=800.0 PL=0
MOVL C00083 V=800.0 PL=0
MOVL C00084 V=800.0 PL=0
MOVL C00085 V=800.0 PL=0
MOVL C00086 V=800.0 PL=0
MOVL C00087 V=800.0 PL=0
MOVL C00088 V=800.0 PL=0
MOVL C00089 V=800.0 PL=0
MOVL C00090 V=800.0 PL=0
MOVL C00091 V=800.0 PL=0
MOVL C00092 V=800.0 PL=0
MOVL C00093 V=800.0 PL=0
MOVL C00094 V=800.0 PL=0
MOVL C00095 V=800.0 PL=0
MOVL C00096 V=800.0 PL=0
MOVL C00097 V=800.0 PL=0
MOVL C00098 V=800.0 PL=0
MOVL C00099 V=800.0 PL=0
MOVL C00100 V=800.0 PL=0
MOVL C00101 V=800.0 PL=0
MOVL C00102 V=800.0 PL=0
MOVL C00103 V=800.0 PL=0
MOVL C00104 V=800.0 PL=0
MOVL C00105 V=800.0 PL=0
MOVL C00106 V=800.0 PL=0
MOVL C00107 V=800.0 PL=0
MOVL C00108 V=800.0 PL=0
MOVL C00109 V=800.0 PL=0
MOVL C00110 V=800.0 PL=0
MOVL C00111 V=800.0 PL=0
MOVL C00112 V=800.0 PL=0
MOVL C00113 V=800.0 PL=0
MOVL C00114 V=800.0 PL=0
MOVL C00115 V=800.0 PL=0
MOVL C00116 V=800.0 PL=0
MOVL C00117 V=800.0 PL=0
MOVL C00118 V=800.0 PL=0
MOVL C00119 V=800.0 PL=0
MOVL C00120 V=800.0 PL=0
MOVL C00121 V=800.0 PL=0
MOVL C00122 V=800.0 PL=0
MOVL C00123 V=800.0 PL=0
MOVL C00124 V=800.0 PL=0
MOVL C00125 V=800.0 PL=0
MOVL C00126 V=800.0 PL=0
MOVL C00127 V=800.0 PL=0
MOVL C00128 V=800.0 PL=0
MOVL C00129 V=800.0 PL=0
MOVL C00130 V=800.0 PL=0
MOVL C00131 V=800.0 PL=0
MOVL C00132 V=800.0 PL=0
MOVL C00133 V=800.0 PL=0
MOVL C00134 V=800.0 PL=0
MOVL C00135 V=800.0 PL=0
MOVL C00136 V=800.0 PL=0
MOVL C00137 V=800.0 PL=0
MOVL C00138 V=800.0 PL=0
MOVL C00139 V=800.0 PL=0
MOVL C00140 V=800.0 PL=0
MOVL C00141 V=800.0 PL=0
MOVL C00142 V=800.0 PL=0
MOVL C00143 V=800.0 PL=0
MOVL C00144 V=800.0 PL=0
MOVL C00145 V=800.0 PL=0
MOVL C00146 V=800.0 PL=0
MOVL C00147 V=800.0 PL=0
MOVL C00148 V=800.0 PL=0
MOVL C00149 V=800.0 PL=0
MOVL C00150 V=800.0 PL=0
MOVL C00151 V=800.0 PL=0
MOVL C00152 V=800.0 PL=0
MOVL C00153 V=800.0 PL=0
MOVL C00154 V=800.0 PL=0
MOVL C00155 V=800.0 PL=0
MOVL C00156 V=800.0 PL=0
MOVL C00157 V=800.0 PL=0
MOVL C00158 V=800.0 PL=0
MOVL C00159 V=800.0 PL=0
MOVL C00160 V=800.0 PL=0
MOVL C00161 V=800.0 PL=0
MOVL C00162 V=800.0 PL=0
MOVL C00163 V=800.0 PL=0
MOVL C00164 V=800.0 PL=0
MOVL C00165 V=800.0 PL=0
MOVL C00166 V=800.0 PL=0
MOVL C00167 V=800.0 PL=0
MOVL C00168 V=800.0 PL=0
MOVL C00169 V=800.0 PL=0
MOVL C00170 V=800.0 PL=0
MOVL C00171 V=800.0 PL=0
MOVL C00172 V=800.0 PL=0
MOVL C00173 V=800.0 PL=0
MOVL C00174 V=800.0 PL=0
MOVL C00175 V=800.0 PL=0
MOVL C00176 V=800.0 PL=0
MOVL C00177 V=800.0 PL=0
MOVL C00178 V=800.0 PL=0
MOVL C00179 V=800.0 PL=0
MOVL C00180 V=800.0 PL=0
MOVL C00181 V=800.0 PL=0
MOVL C00182 V=800.0 PL=0
MOVL C00183 V=800.0 PL=0
MOVL C00184 V=800.0 PL=0
MOVL C00185 V=800.0 PL=0
MOVL C00186 V=800.0 PL=0
MOVL C00187 V=800.0 PL=0
MOVL C00188 V=800.0 PL=0
MOVL C00189 V=800.0 PL=0
MOVL C00190 V=800.0 PL=0
MOVL C00191 V=800.0 PL=0
MOVL C00192 V=800.0 PL=0
MOVL C00193 V=800.0 PL=0
MOVL C00194 V=800.0 PL=0
MOVL C00195 V=800.0 PL=0
MOVL C00196 V=800.0 PL=0
MOVL C00197 V=800.0 PL=0
MOVL C00198 V=800.0 PL=0
MOVL C00199 V=800.0 PL=0
MOVL C00200 V=800.0 PL=0
MOVL C00201 V=800.0 PL=0
MOVL C00202 V=800.0 PL=0
MOVL C00203 V=800.0 PL=0
MOVL C00204 V=800.0 PL=0
MOVL C00205 V=800.0 PL=0
MOVL C00206 V=800.0 PL=0
MOVL C00207 V=800.0 PL=0
MOVL C00208 V=800.0 PL=0
MOVL C00209 V=800.0 PL=0
MOVL C00210 V=800.0 PL=0
MOVL C00211 V=800.0 PL=0
MOVL C00212 V=800.0 PL=0
MOVL C00213 V=800.0 PL=0
MOVL C00214 V=800.0 PL=0
MOVL C00215 V=800.0 PL=0
MOVL C00216 V=800.0 PL=0
MOVL C00217 V=800.0 PL=0
MOVL C00218 V=800.0 PL=0
MOVL C00219 V=800.0 PL=0
MOVL C00220 V=800.0 PL=0
MOVL C00221 V=800.0 PL=0
MOVL C00222 V=800.0 PL=0
MOVL C00223 V=800.0 PL=0
MOVL C00224 V=800.0 PL=0
MOVL C00225 V=800.0 PL=0
MOVL C00226 V=800.0 PL=0
MOVL C00227 V=800.0 PL=0
MOVL C00228 V=800.0 PL=0
MOVL C00229 V=800.0 PL=0
MOVL C00230 V=800.0 PL=0
MOVL C00231 V=800.0 PL=0
MOVL C00232 V=800.0 PL=0
MOVL C00233 V=800.0 PL=0
MOVL C00234 V=800.0 PL=0
MOVL C00235 V=800.0 PL=0
MOVL C00236 V=800.0 PL=0
MOVL C00237 V=800.0 PL=0
MOVL C00238 V=800.0 PL=0
MOVL C00239 V=800.0 PL=0
MOVL C00240 V=800.0 PL=0
MOVL C00241 V=800.0 PL=0
MOVL C00242 V=800.0 PL=0
MOVL C00243 V=800.0 PL=0
MOVL C00244 V=800.0 PL=0
MOVL C00245 V=800.0 PL=0
MOVL C00246 V=800.0 PL=0
MOVL C00247 V=800.0 PL=0
MOVL C00248 V=800.0 PL=0
MOVL C00249 V=800.0 PL=0
MOVL C00250 V=800.0 PL=0
MOVL C00251 V=800.0 PL=0
MOVL C00252 V=800.0 PL=0
MOVL C00253 V=800.0 PL=0
MOVL C00254 V=800.0 PL=0
MOVL C00255 V=800.0 PL=0
MOVL C00256 V=800.0 PL=0
MOVL C00257 V=800.0 PL=0
MOVL C00258 V=800.0 PL=0
MOVL C00259 V=800.0 PL=0
MOVL C00260 V=800.0 PL=0
MOVL C00261 V=800.0 PL=0
MOVL C00262 V=800.0 PL=0
MOVL C00263 V=800.0 PL=0
MOVL C00264 V=800.0 PL=0
MOVL C00265 V=800.0 PL=0
MOVL C00266 V=800.0 PL=0
MOVL C00267 V=800.0 PL=0
MOVL C00268 V=800.0 PL=0
MOVL C00269 V=800.0 PL=0
MOVL C00270 V=800.0 PL=0
MOVL C00271 V=800.0 PL=0
MOVL C00272 V=800.0 PL=0
MOVL C00273 V=800.0 PL=0
MOVL C00274 V=800.0 PL=0
MOVL C00275 V=800.0 PL=0
MOVL C00276 V=800.0 PL=0
MOVL C00277 V=800.0 PL=0
MOVL C00278 V=800.0 PL=0
MOVL C00279 V=800.0 PL=0
MOVL C00280 V=800.0 PL=0
MOVL C00281 V=800.0 PL=0
MOVL C00282 V=800.0 PL=0
MOVL C00283 V=800.0 PL=0
MOVL C00284 V=800.0 PL=0
MOVL C00285 V=800.0 PL=0
MOVL C00286 V=800.0 PL=0
MOVL C00287 V=800.0 PL=0
MOVL C00288 V=800.0 PL=0
MOVL C00289 V=800.0 PL=0
MOVL C00290 V=800.0 PL=0
MOVL C00291 V=800.0 PL=0
MOVL C00292 V=800.0 PL=0
MOVL C00293 V=800.0 PL=0
MOVL C00294 V=800.0 PL=0
MOVL C00295 V=800.0 PL=0
MOVL C00296 V=800.0 PL=0
MOVL C00297 V=800.0 PL=0
MOVL C00298 V=800.0 PL=0
MOVL C00299 V=800.0 PL=0
MOVL C00300 V=800.0 PL=0
MOVL C00301 V=800.0 PL=0
MOVL C00302 V=800.0 PL=0
MOVL C00303 V=800.0 PL=0
MOVL C00304 V=800.0 PL=0
MOVL C00305 V=800.0 PL=0
MOVL C00306 V=800.0 PL=0
MOVL C00307 V=800.0 PL=0
MOVL C00308 V=800.0 PL=0
MOVL C00309 V=800.0 PL=0
MOVL C00310 V=800.0 PL=0
MOVL C00311 V=800.0 PL=0
MOVL C00312 V=800.0 PL=0
MOVL C00313 V=800.0 PL=0
MOVL C00314 V=800.0 PL=0
MOVL C00315 V=800.0 PL=0
MOVL C00316 V=800.0 PL=0
MOVL C00317 V=800.0 PL=0
MOVL C00318 V=800.0 PL=0
MOVL C00319 V=800.0 PL=0
MOVL C00320 V=800.0 PL=0
MOVL C00321 V=800.0 PL=0
MOVL C00322 V=800.0 PL=0
MOVL C00323 V=800.0 PL=0
MOVL C00324 V=800.0 PL=0
MOVL C00325 V=800.0 PL=0
MOVL C00326 V=800.0 PL=0
MOVL C00327 V=800.0 PL=0
MOVL C00328 V=800.0 PL=0
MOVL C00329 V=800.0 PL=0
MOVL C00330 V=800.0 PL=0
MOVL C00331 V=800.0 PL=0
MOVL C00332 V=800.0 PL=0
MOVL C00333 V=800.0 PL=0
MOVL C00334 V=800.0 PL=0
MOVL C00335 V=800.0 PL=0
MOVL C00336 V=800.0 PL=0
MOVL C00337 V=800.0 PL=0
MOVL C00338 V=800.0 PL=0
MOVL C00339 V=800.0 PL=0
MOVL C00340 V=800.0 PL=0
MOVL C00341 V=800.0 PL=0
MOVL C00342 V=800.0 PL=0
MOVL C00343 V=800.0 PL=0
MOVL C00344 V=800.0 PL=0
MOVL C00345 V=800.0 PL=0
MOVL C00346 V=800.0 PL=0
MOVL C00347 V=800.0 PL=0
MOVL C00348 V=800.0 PL=0
MOVL C00349 V=800.0 PL=0
MOVL C00350 V=800.0 PL=0
MOVL C00351 V=800.0 PL=0
MOVL C00352 V=800.0 PL=0
MOVL C00353 V=800.0 PL=0
MOVL C00354 V=800.0 PL=0
MOVL C00355 V=800.0 PL=0
MOVL C00356 V=800.0 PL=0
MOVL C00357 V=800.0 PL=0
MOVL C00358 V=800.0 PL=0
MOVL C00359 V=800.0 PL=0
MOVL C00360 V=800.0 PL=0
MOVL C00361 V=800.0 PL=0
MOVL C00362 V=800.0 PL=0
MOVL C00363 V=800.0 PL=0
MOVL C00364 V=800.0 PL=0
MOVL C00365 V=800.0 PL=0
MOVL C00366 V=800.0 PL=0
MOVL C00367 V=800.0 PL=0
MOVL C00368 V=800.0 PL=0
MOVL C00369 V=800.0 PL=0
MOVL C00370 V=800.0 PL=0
MOVL C00371 V=800.0 PL=0
MOVL C00372 V=800.0 PL=0
MOVL C00373 V=800.0 PL=0
MOVL C00374 V=800.0 PL=0
MOVL C00375 V=800.0 PL=0
MOVL C00376 V=800.0 PL=0
MOVL C00377 V=800.0 PL=0
MOVL C00378 V=800.0 PL=0
MOVL C00379 V=800.0 PL=0
MOVL C00380 V=800.0 PL=0
MOVL C00381 V=800.0 PL=0
MOVL C00382 V=800.0 PL=0
MOVL C00383 V=800.0 PL=0
MOVL C00384 V=800.0 PL=0
MOVL C00385 V=800.0 PL=0
MOVL C00386 V=800.0 PL=0
MOVL C00387 V=800.0 PL=0
MOVL C00388 V=800.0 PL=0
MOVL C00389 V=800.0 PL=0
MOVL C00390 V=800.0 PL=0
MOVL C00391 V=800.0 PL=0
MOVL C00392 V=800.0 PL=0
MOVL C00393 V=800.0 PL=0
MOVL C00394 V=800.0 PL=0
MOVL C00395 V=800.0 PL=0
MOVL C00396 V=800.0 PL=0
MOVL C00397 V=800.0 PL=0
MOVL C00398 V=800.0 PL=0
MOVL C00399 V=800.0 PL=0
MOVL C00400 V=800.0 PL=0
MOVL C00401 V=800.0 PL=0
MOVL C00402 V=800.0 PL=0
MOVL C00403 V=800.0 PL=0
MOVL C00404 V=800.0 PL=0
MOVL C00405 V=800.0 PL=0
MOVL C00406 V=800.0 PL=0
MOVL C00407 V=800.0 PL=0
MOVL C00408 V=800.0 PL=0
MOVL C00409 V=800.0 PL=0
MOVL C00410 V=800.0 PL=0
MOVL C00411 V=800.0 PL=0
MOVL C00412 V=800.0 PL=0
MOVL C00413 V=800.0 PL=0
MOVL C00414 V=800.0 PL=0
MOVL C00415 V=800.0 PL=0
MOVL C00416 V=800.0 PL=0
MOVL C00417 V=800.0 PL=0
MOVL C00418 V=800.0 PL=0
MOVL C00419 V=800.0 PL=0
MOVL C00420 V=800.0 PL=0
MOVL C00421 V=800.0 PL=0
MOVL C00422 V=800.0 PL=0
MOVL C00423 V=800.0 PL=0
MOVL C00424 V=800.0 PL=0
MOVL C00425 V=800.0 PL=0
MOVL C00426 V=800.0 PL=0
MOVL C00427 V=800.0 PL=0
MOVL C00428 V=800.0 PL=0
MOVL C00429 V=800.0 PL=0
MOVL C00430 V=800.0 PL=0
MOVL C00431 V=800.0 PL=0
MOVL C00432 V=800.0 PL=0
MOVL C00433 V=800.0 PL=0
MOVL C00434 V=800.0 PL=0
MOVL C00435 V=800.0 PL=0
MOVL C00436 V=800.0 PL=0
MOVL C00437 V=800.0 PL=0
MOVL C00438 V=800.0 PL=0
MOVL C00439 V=800.0 PL=0
MOVL C00440 V=800.0 PL=0
MOVL C00441 V=800.0 PL=0
MOVL C00442 V=800.0 PL=0
MOVL C00443 V=800.0 PL=0
MOVL C00444 V=800.0 PL=0
MOVL C00445 V=800.0 PL=0
MOVL C00446 V=800.0 PL=0
MOVL C00447 V=800.0 PL=0
MOVL C00448 V=800.0 PL=0
MOVL C00449 V=800.0 PL=0
MOVL C00450 V=800.0 PL=0
MOVL C00451 V=800.0 PL=0
MOVL C00452 V=800.0 PL=0
MOVL C00453 V=800.0 PL=0
MOVL C00454 V=800.0 PL=0
MOVL C00455 V=800.0 PL=0
MOVL C00456 V=800.0 PL=0
MOVL C00457 V=800.0 PL=0
MOVL C00458 V=800.0 PL=0
MOVL C00459 V=800.0 PL=0
MOVL C00460 V=800.0 PL=0
MOVL C00461 V=800.0 PL=0
MOVL C00462 V=800.0 PL=0
MOVL C00463 V=800.0 PL=0
MOVL C00464 V=800.0 PL=0
MOVL C00465 V=800.0 PL=0
MOVL C00466 V=800.0 PL=0
MOVL C00467 V=800.0 PL=0
MOVL C00468 V=800.0 PL=0
MOVL C00469 V=800.0 PL=0
MOVL C00470 V=800.0 PL=0
MOVL C00471 V=800.0 PL=0
MOVL C00472 V=800.0 PL=0
MOVL C00473 V=800.0 PL=0
MOVL C00474 V=800.0 PL=0
MOVL C00475 V=800.0 PL=0
MOVL C00476 V=800.0 PL=0
MOVL C00477 V=800.0 PL=0
MOVL C00478 V=800.0 PL=0
MOVL C00479 V=800.0 PL=0
MOVL C00480 V=800.0 PL=0
MOVL C00481 V=800.0 PL=0
MOVL C00482 V=800.0 PL=0
MOVL C00483 V=800.0 PL=0
MOVL C00484 V=800.0 PL=0
MOVL C00485 V=800.0 PL=0
MOVL C00486 V=800.0 PL=0
MOVL C00487 V=800.0 PL=0
MOVL C00488 V=800.0 PL=0
MOVL C00489 V=800.0 PL=0
MOVL C00490 V=800.0 PL=0
MOVL C00491 V=800.0 PL=0
MOVL C00492 V=800.0 PL=0
MOVL C00493 V=800.0 PL=0
MOVL C00494 V=800.0 PL=0
MOVL C00495 V=800.0 PL=0
MOVL C00496 V=800.0 PL=0
MOVL C00497 V=800.0 PL=0
MOVL C00498 V=800.0 PL=0
MOVL C00499 V=800.0 PL=0
MOVL C00500 V=800.0 PL=0
MOVL C00501 V=800.0 PL=0
MOVL C00502 V=800.0 PL=0
MOVL C00503 V=800.0 PL=0
MOVL C00504 V=800.0 PL=0
MOVL C00505 V=800.0 PL=0
MOVL C00506 V=800.0 PL=0
MOVL C00507 V=800.0 PL=0
MOVL C00508 V=800.0 PL=0
MOVL C00509 V=800.0 PL=0
MOVL C00510 V=800.0 PL=0
MOVL C00511 V=800.0 PL=0
MOVL C00512 V=800.0 PL=0
MOVL C00513 V=800.0 PL=0
MOVL C00514 V=800.0 PL=0
MOVL C00515 V=800.0 PL=0
MOVL C00516 V=800.0 PL=0
MOVL C00517 V=800.0 PL=0
MOVL C00518 V=800.0 PL=0
MOVL C00519 V=800.0 PL=0
MOVL C00520 V=800.0 PL=0
MOVL C00521 V=800.0 PL=0
MOVL C00522 V=800.0 PL=0
MOVL C00523 V=800.0 PL=0
MOVL C00524 V=800.0 PL=0
MOVL C00525 V=800.0 PL=0
MOVL C00526 V=800.0 PL=0
MOVL C00527 V=800.0 PL=0
MOVL C00528 V=800.0 PL=0
MOVL C00529 V=800.0 PL=0
MOVL C00530 V=800.0 PL=0
MOVL C00531 V=800.0 PL=0
MOVL C00532 V=800.0 PL=0
MOVL C00533 V=800.0 PL=0
MOVL C00534 V=800.0 PL=0
MOVL C00535 V=800.0 PL=0
MOVL C00536 V=800.0 PL=0
MOVL C00537 V=800.0 PL=0
MOVL C00538 V=800.0 PL=0
MOVL C00539 V=800.0 PL=0
MOVL C00540 V=800.0 PL=0
MOVL C00541 V=800.0 PL=0
MOVL C00542 V=800.0 PL=0
MOVL C00543 V=800.0 PL=0
MOVL C00544 V=800.0 PL=0
MOVL C00545 V=800.0 PL=0
MOVL C00546 V=800.0 PL=0
MOVL C00547 V=800.0 PL=0
MOVL C00548 V=800.0 PL=0
MOVL C00549 V=800.0 PL=0
MOVL C00550 V=800.0 PL=0
MOVL C00551 V=800.0 PL=0
MOVL C00552 V=800.0 PL=0
MOVL C00553 V=800.0 PL=0
MOVL C00554 V=800.0 PL=0
MOVL C00555 V=800.0 PL=0
MOVL C00556 V=800.0 PL=0
MOVL C00557 V=800.0 PL=0
MOVL C00558 V=800.0 PL=0
MOVL C00559 V=800.0 PL=0
MOVL C00560 V=800.0 PL=0
MOVL C00561 V=800.0 PL=0
MOVL C00562 V=800.0 PL=0
MOVL C00563 V=800.0 PL=0
MOVL C00564 V=800.0 PL=0
MOVL C00565 V=800.0 PL=0
MOVL C00566 V=800.0 PL=0
MOVL C00567 V=800.0 PL=0
MOVL C00568 V=800.0 PL=0
MOVL C00569 V=800.0 PL=0
MOVL C00570 V=800.0 PL=0
MOVL C00571 V=800.0 PL=0
MOVL C00572 V=800.0 PL=0
MOVL C00573 V=800.0 PL=0
MOVL C00574 V=800.0 PL=0
MOVL C00575 V=800.0 PL=0
MOVL C00576 V=800.0 PL=0
MOVL C00577 V=800.0 PL=0
MOVL C00578 V=800.0 PL=0
MOVL C00579 V=800.0 PL=0
MOVL C00580 V=800.0 PL=0
MOVL C00581 V=800.0 PL=0
MOVL C00582 V=800.0 PL=0
MOVL C00583 V=800.0 PL=0
MOVL C00584 V=800.0 PL=0
MOVL C00585 V=800.0 PL=0
MOVL C00586 V=800.0 PL=0
MOVL C00587 V=800.0 PL=0
MOVL C00588 V=800.0 PL=0
MOVL C00589 V=800.0 PL=0
MOVL C00590 V=800.0 PL=0
MOVL C00591 V=800.0 PL=0
MOVL C00592 V=800.0 PL=0
MOVL C00593 V=800.0 PL=0
MOVL C00594 V=800.0 PL=0
MOVL C00595 V=800.0 PL=0
MOVL C00596 V=800.0 PL=0
MOVL C00597 V=800.0 PL=0
MOVL C00598 V=800.0 PL=0
MOVL C00599 V=800.0 PL=0
MOVL C00600 V=800.0 PL=0
MOVL C00601 V=800.0 PL=0
MOVL C00602 V=800.0 PL=0
MOVL C00603 V=800.0 PL=0
MOVL C00604 V=800.0 PL=0
MOVL C00605 V=800.0 PL=0
MOVL C00606 V=800.0 PL=0
MOVL C00607 V=800.0 PL=0
MOVL C00608 V=800.0 PL=0
MOVL C00609 V=800.0 PL=0
MOVL C00610 V=800.0 PL=0
MOVL C00611 V=800.0 PL=0
MOVL C00612 V=800.0 PL=0
MOVL C00613 V=800.0 PL=0
MOVL C00614 V=800.0 PL=0
MOVL C00615 V=800.0 PL=0
MOVL C00616 V=800.0 PL=0
MOVL C00617 V=800.0 PL=0
MOVL C00618 V=800.0 PL=0
MOVL C00619 V=800.0 PL=0
MOVL C00620 V=800.0 PL=0
MOVL C00621 V=800.0 PL=0
MOVL C00622 V=800.0 PL=0
MOVL C00623 V=800.0 PL=0
MOVL C00624 V=800.0 PL=0
MOVL C00625 V=800.0 PL=0
MOVL C00626 V=800.0 PL=0
MOVL C00627 V=800.0 PL=0
MOVL C00628 V=800.0 PL=0
MOVL C00629 V=800.0 PL=0
MOVL C00630 V=800.0 PL=0
MOVL C00631 V=800.0 PL=0
MOVL C00632 V=800.0 PL=0
MOVL C00633 V=800.0 PL=0
MOVL C00634 V=800.0 PL=0
MOVL C00635 V=800.0 PL=0
MOVL C00636 V=800.0 PL=0
MOVL C00637 V=800.0 PL=0
MOVL C00638 V=800.0 PL=0
MOVL C00639 V=800.0 PL=0
MOVL C00640 V=800.0 PL=0
MOVL C00641 V=800.0 PL=0
MOVL C00642 V=800.0 PL=0
MOVL C00643 V=800.0 PL=0
MOVL C00644 V=800.0 PL=0
MOVL C00645 V=800.0 PL=0
MOVL C00646 V=800.0 PL=0
MOVL C00647 V=800.0 PL=0
MOVL C00648 V=800.0 PL=0
MOVL C00649 V=800.0 PL=0
MOVL C00650 V=800.0 PL=0
MOVL C00651 V=800.0 PL=0
MOVL C00652 V=800.0 PL=0
MOVL C00653 V=800.0 PL=0
MOVL C00654 V=800.0 PL=0
MOVL C00655 V=800.0 PL=0
MOVL C00656 V=800.0 PL=0
MOVL C00657 V=800.0 PL=0
MOVL C00658 V=800.0 PL=0
MOVL C00659 V=800.0 PL=0
MOVL C00660 V=800.0 PL=0
MOVL C00661 V=800.0 PL=0
MOVL C00662 V=800.0 PL=0
MOVL C00663 V=800.0 PL=0
MOVL C00664 V=800.0 PL=0
MOVL C00665 V=800.0 PL=0
MOVL C00666 V=800.0 PL=0
MOVL C00667 V=800.0 PL=0
MOVL C00668 V=800.0 PL=0
MOVL C00669 V=800.0 PL=0
MOVL C00670 V=800.0 PL=0
MOVL C00671 V=800.0 PL=0
MOVL C00672 V=800.0 PL=0
MOVL C00673 V=800.0 PL=0
MOVL C00674 V=800.0 PL=0
MOVL C00675 V=800.0 PL=0
MOVL C00676 V=800.0 PL=0
MOVL C00677 V=800.0 PL=0
MOVL C00678 V=800.0 PL=0
MOVL C00679 V=800.0 PL=0
MOVL C00680 V=800.0 PL=0
MOVL C00681 V=800.0 PL=0
MOVL C00682 V=800.0 PL=0
MOVL C00683 V=800.0 PL=0
MOVL C00684 V=800.0 PL=0
MOVL C00685 V=800.0 PL=0
MOVL C00686 V=800.0 PL=0
MOVL C00687 V=800.0 PL=0
MOVL C00688 V=800.0 PL=0
MOVL C00689 V=800.0 PL=0
MOVL C00690 V=800.0 PL=0
MOVL C00691 V=800.0 PL=0
MOVL C00692 V=800.0 PL=0
MOVL C00693 V=800.0 PL=0
MOVL C00694 V=800.0 PL=0
MOVL C00695 V=800.0 PL=0
MOVL C00696 V=800.0 PL=0
MOVL C00697 V=800.0 PL=0
MOVL C00698 V=800.0 PL=0
MOVL C00699 V=800.0 PL=0
MOVL C00700 V=800.0 PL=0
MOVL C00701 V=800.0 PL=0
MOVL C00702 V=800.0 PL=0
MOVL C00703 V=800.0 PL=0
MOVL C00704 V=800.0 PL=0
MOVL C00705 V=800.0 PL=0
MOVL C00706 V=800.0 PL=0
MOVL C00707 V=800.0 PL=0
MOVL C00708 V=800.0 PL=0
MOVL C00709 V=800.0 PL=0
MOVL C00710 V=800.0 PL=0
MOVL C00711 V=800.0 PL=0
MOVL C00712 V=800.0 PL=0
MOVL C00713 V=800.0 PL=0
MOVL C00714 V=800.0 PL=0
MOVL C00715 V=800.0 PL=0
MOVL C00716 V=800.0 PL=0
MOVL C00717 V=800.0 PL=0
MOVL C00718 V=800.0 PL=0
MOVL C00719 V=800.0 PL=0
MOVL C00720 V=800.0 PL=0
MOVL C00721 V=800.0 PL=0
MOVL C00722 V=800.0 PL=0
MOVL C00723 V=800.0 PL=0
MOVL C00724 V=800.0 PL=0
MOVL C00725 V=800.0 PL=0
MOVL C00726 V=800.0 PL=0
MOVL C00727 V=800.0 PL=0
MOVL C00728 V=800.0 PL=0
MOVL C00729 V=800.0 PL=0
MOVL C00730 V=800.0 PL=0
MOVL C00731 V=800.0 PL=0
MOVL C00732 V=800.0 PL=0
MOVL C00733 V=800.0 PL=0
MOVL C00734 V=800.0 PL=0
MOVL C00735 V=800.0 PL=0
MOVL C00736 V=800.0 PL=0
MOVL C00737 V=800.0 PL=0
MOVL C00738 V=800.0 PL=0
MOVL C00739 V=800.0 PL=0
MOVL C00740 V=800.0 PL=0
MOVL C00741 V=800.0 PL=0
MOVL C00742 V=800.0 PL=0
MOVL C00743 V=800.0 PL=0
MOVL C00744 V=800.0 PL=0
MOVL C00745 V=800.0 PL=0
MOVL C00746 V=800.0 PL=0
MOVL C00747 V=800.0 PL=0
MOVL C00748 V=800.0 PL=0
MOVL C00749 V=800.0 PL=0
MOVL C00750 V=800.0 PL=0
MOVL C00751 V=800.0 PL=0
MOVL C00752 V=800.0 PL=0
MOVL C00753 V=800.0 PL=0
MOVL C00754 V=800.0 PL=0
MOVL C00755 V=800.0 PL=0
MOVL C00756 V=800.0 PL=0
MOVL C00757 V=800.0 PL=0
MOVL C00758 V=800.0 PL=0
MOVL C00759 V=800.0 PL=0
MOVL C00760 V=800.0 PL=0
MOVL C00761 V=800.0 PL=0
MOVL C00762 V=800.0 PL=0
MOVL C00763 V=800.0 PL=0
MOVL C00764 V=800.0 PL=0
MOVL C00765 V=800.0 PL=0
MOVL C00766 V=800.0 PL=0
MOVL C00767 V=800.0 PL=0
MOVL C00768 V=800.0 PL=0
MOVL C00769 V=800.0 PL=0
MOVL C00770 V=800.0 PL=0
MOVL C00771 V=800.0 PL=0
MOVL C00772 V=800.0 PL=0
MOVL C00773 V=800.0 PL=0
MOVL C00774 V=800.0 PL=0
MOVL C00775 V=800.0 PL=0
MOVL C00776 V=800.0 PL=0
MOVL C00777 V=800.0 PL=0
MOVL C00778 V=800.0 PL=0
MOVL C00779 V=800.0 PL=0
MOVL C00780 V=800.0 PL=0
MOVL C00781 V=800.0 PL=0
MOVL C00782 V=800.0 PL=0
MOVL C00783 V=800.0 PL=0
MOVL C00784 V=800.0 PL=0
MOVL C00785 V=800.0 PL=0
MOVL C00786 V=800.0 PL=0
MOVL C00787 V=800.0 PL=0
MOVL C00788 V=800.0 PL=0
MOVL C00789 V=800.0 PL=0
MOVL C00790 V=800.0 PL=0
MOVL C00791 V=800.0 PL=0
MOVL C00792 V=800.0 PL=0
MOVL C00793 V=800.0 PL=0
MOVL C00794 V=800.0 PL=0
MOVL C00795 V=800.0 PL=0
MOVL C00796 V=800.0 PL=0
MOVL C00797 V=800.0 PL=0
MOVL C00798 V=800.0 PL=0
MOVL C00799 V=800.0 PL=0
MOVL C00800 V=800.0 PL=0
MOVL C00801 V=800.0 PL=0
MOVL C00802 V=800.0 PL=0
MOVL C00803 V=800.0 PL=0
MOVL C00804 V=800.0 PL=0
MOVL C00805 V=800.0 PL=0
MOVL C00806 V=800.0 PL=0
MOVL C00807 V=800.0 PL=0
MOVL C00808 V=800.0 PL=0
MOVL C00809 V=800.0 PL=0
MOVL C00810 V=800.0 PL=0
MOVL C00811 V=800.0 PL=0
MOVL C00812 V=800.0 PL=0
MOVL C00813 V=800.0 PL=0
MOVL C00814 V=800.0 PL=0
MOVL C00815 V=800.0 PL=0
MOVL C00816 V=800.0 PL=0
MOVL C00817 V=800.0 PL=0
MOVL C00818 V=800.0 PL=0
MOVL C00819 V=800.0 PL=0
MOVL C00820 V=800.0 PL=0
MOVL C00821 V=800.0 PL=0
MOVL C00822 V=800.0 PL=0
MOVL C00823 V=800.0 PL=0
MOVL C00824 V=800.0 PL=0
MOVL C00825 V=800.0 PL=0
MOVL C00826 V=800.0 PL=0
MOVL C00827 V=800.0 PL=0
MOVL C00828 V=800.0 PL=0
MOVL C00829 V=800.0 PL=0
MOVL C00830 V=800.0 PL=0
MOVL C00831 V=800.0 PL=0
MOVL C00832 V=800.0 PL=0
MOVL C00833 V=800.0 PL=0
MOVL C00834 V=800.0 PL=0
MOVL C00835 V=800.0 PL=0
MOVL C00836 V=800.0 PL=0
MOVL C00837 V=800.0 PL=0
MOVL C00838 V=800.0 PL=0
MOVL C00839 V=800.0 PL=0
MOVL C00840 V=800.0 PL=0
MOVL C00841 V=800.0 PL=0
MOVL C00842 V=800.0 PL=0
MOVL C00843 V=800.0 PL=0
MOVL C00844 V=800.0 PL=0
MOVL C00845 V=800.0 PL=0
MOVL C00846 V=800.0 PL=0
MOVL C00847 V=800.0 PL=0
MOVL C00848 V=800.0 PL=0
MOVL C00849 V=800.0 PL=0
MOVL C00850 V=800.0 PL=0
MOVL C00851 V=800.0 PL=0
MOVL C00852 V=800.0 PL=0
MOVL C00853 V=800.0 PL=0
MOVL C00854 V=800.0 PL=0
MOVL C00855 V=800.0 PL=0
MOVL C00856 V=800.0 PL=0
MOVL C00857 V=800.0 PL=0
MOVL C00858 V=800.0 PL=0
MOVL C00859 V=800.0 PL=0
MOVL C00860 V=800.0 PL=0
MOVL C00861 V=800.0 PL=0
MOVL C00862 V=800.0 PL=0
MOVL C00863 V=800.0 PL=0
MOVL C00864 V=800.0 PL=0
MOVL C00865 V=800.0 PL=0
MOVL C00866 V=800.0 PL=0
MOVL C00867 V=800.0 PL=0
MOVL C00868 V=800.0 PL=0
MOVL C00869 V=800.0 PL=0
MOVL C00870 V=800.0 PL=0
MOVL C00871 V=800.0 PL=0
MOVL C00872 V=800.0 PL=0
MOVL C00873 V=800.0 PL=0
MOVL C00874 V=800.0 PL=0
MOVL C00875 V=800.0 PL=0
MOVL C00876 V=800.0 PL=0
MOVL C00877 V=800.0 PL=0
MOVL C00878 V=800.0 PL=0
MOVL C00879 V=800.0 PL=0
MOVL C00880 V=800.0 PL=0
MOVL C00881 V=800.0 PL=0
MOVL C00882 V=800.0 PL=0
MOVL C00883 V=800.0 PL=0
MOVL C00884 V=800.0 PL=0
MOVL C00885 V=800.0 PL=0
MOVL C00886 V=800.0 PL=0
MOVL C00887 V=800.0 PL=0
MOVL C00888 V=800.0 PL=0
MOVL C00889 V=800.0 PL=0
MOVL C00890 V=800.0 PL=0
MOVL C00891 V=800.0 PL=0
MOVL C00892 V=800.0 PL=0
MOVL C00893 V=800.0 PL=0
MOVL C00894 V=800.0 PL=0
MOVL C00895 V=800.0 PL=0
MOVL C00896 V=800.0 PL=0
MOVL C00897 V=800.0 PL=0
MOVL C00898 V=800.0 PL=0
MOVL C00899 V=800.0 PL=0
MOVL C00900 V=800.0 PL=0
MOVL C00901 V=800.0 PL=0
MOVL C00902 V=800.0 PL=0
MOVL C00903 V=800.0 PL=0
MOVL C00904 V=800.0 PL=0
MOVL C00905 V=800.0 PL=0
MOVL C00906 V=800.0 PL=0
MOVL C00907 V=800.0 PL=0
MOVL C00908 V=800.0 PL=0
MOVL C00909 V=800.0 PL=0
MOVL C00910 V=800.0 PL=0
MOVL C00911 V=800.0 PL=0
MOVL C00912 V=800.0 PL=0
MOVL C00913 V=800.0 PL=0
MOVL C00914 V=800.0 PL=0
MOVL C00915 V=800.0 PL=0
MOVL C00916 V=800.0 PL=0
MOVL C00917 V=800.0 PL=0
MOVL C00918 V=800.0 PL=0
MOVL C00919 V=800.0 PL=0
MOVL C00920 V=800.0 PL=0
MOVL C00921 V=800.0 PL=0
MOVL C00922 V=800.0 PL=0
MOVL C00923 V=800.0 PL=0
MOVL C00924 V=800.0 PL=0
MOVL C00925 V=800.0 PL=0
MOVL C00926 V=800.0 PL=0
MOVL C00927 V=800.0 PL=0
MOVL C00928 V=800.0 PL=0
MOVL C00929 V=800.0 PL=0
MOVL C00930 V=800.0 PL=0
MOVL C00931 V=800.0 PL=0
MOVL C00932 V=800.0 PL=0
MOVL C00933 V=800.0 PL=0
MOVL C00934 V=800.0 PL=0
MOVL C00935 V=800.0 PL=0
MOVL C00936 V=800.0 PL=0
MOVL C00937 V=800.0 PL=0
MOVL C00938 V=800.0 PL=0
MOVL C00939 V=800.0 PL=0
MOVL C00940 V=800.0 PL=0
MOVL C00941 V=800.0 PL=0
MOVL C00942 V=800.0 PL=0
MOVL C00943 V=800.0 PL=0
MOVL C00944 V=800.0 PL=0
MOVL C00945 V=800.0 PL=0
MOVL C00946 V=800.0 PL=0
MOVL C00947 V=800.0 PL=0
MOVL C00948 V=800.0 PL=0
MOVL C00949 V=800.0 PL=0
MOVL C00950 V=800.0 PL=0
MOVL C00951 V=800.0 PL=0
MOVL C00952 V=800.0 PL=0
MOVL C00953 V=800.0 PL=0
MOVL C00954 V=800.0 PL=0
MOVL C00955 V=800.0 PL=0
MOVL C00956 V=800.0 PL=0
MOVL C00957 V=800.0 PL=0
MOVL C00958 V=800.0 PL=0
MOVL C00959 V=800.0 PL=0
MOVL C00960 V=800.0 PL=0
MOVL C00961 V=800.0 PL=0
MOVL C00962 V=800.0 PL=0
MOVL C00963 V=800.0 PL=0
MOVL C00964 V=800.0 PL=0
MOVL C00965 V=800.0 PL=0
MOVL C00966 V=800.0 PL=0
MOVL C00967 V=800.0 PL=0
MOVL C00968 V=800.0 PL=0
MOVL C00969 V=800.0 PL=0
MOVL C00970 V=800.0 PL=0
MOVL C00971 V=800.0 PL=0
MOVL C00972 V=800.0 PL=0
MOVL C00973 V=800.0 PL=0
MOVL C00974 V=800.0 PL=0
MOVL C00975 V=800.0 PL=0
MOVL C00976 V=800.0 PL=0
MOVL C00977 V=800.0 PL=0
MOVL C00978 V=800.0 PL=0
MOVL C00979 V=800.0 PL=0
MOVL C00980 V=800.0 PL=0
MOVL C00981 V=800.0 PL=0
MOVL C00982 V=800.0 PL=0
MOVL C00983 V=800.0 PL=0
MOVL C00984 V=800.0 PL=0
MOVL C00985 V=800.0 PL=0
MOVL C00986 V=800.0 PL=0
MOVL C00987 V=800.0 PL=0
MOVL C00988 V=800.0 PL=0
MOVL C00989 V=800.0 PL=0
MOVL C00990 V=800.0 PL=0
MOVL C00991 V=800.0 PL=0
MOVL C00992 V=800.0 PL=0
MOVL C00993 V=800.0 PL=0
MOVL C00994 V=800.0 PL=0
MOVL C00995 V=800.0 PL=0
MOVL C00996 V=800.0 PL=0
MOVL C00997 V=800.0 PL=0
MOVL C00998 V=800.0 PL=0
MOVL C00999 V=800.0 PL=0
MOVL C01000 V=800.0 PL=0
MOVL C01001 V=800.0 PL=0
MOVL C01002 V=800.0 PL=0
MOVL C01003 V=800.0 PL=0
MOVL C01004 V=800.0 PL=0
MOVL C01005 V=800.0 PL=0
MOVL C01006 V=800.0 PL=0
MOVL C01007 V=800.0 PL=0
MOVL C01008 V=800.0 PL=0
MOVL C01009 V=800.0 PL=0
MOVL C01010 V=800.0 PL=0
MOVL C01011 V=800.0 PL=0
MOVL C01012 V=800.0 PL=0
MOVL C01013 V=800.0 PL=0
MOVL C01014 V=800.0 PL=0
MOVL C01015 V=800.0 PL=0
MOVL C01016 V=800.0 PL=0
MOVL C01017 V=800.0 PL=0
MOVL C01018 V=800.0 PL=0
MOVL C01019 V=800.0 PL=0
MOVL C01020 V=800.0 PL=0
MOVL C01021 V=800.0 PL=0
MOVL C01022 V=800.0 PL=0
MOVL C01023 V=800.0 PL=0
MOVL C01024 V=800.0 PL=0
MOVL C01025 V=800.0 PL=0
MOVL C01026 V=800.0 PL=0
MOVL C01027 V=800.0 PL=0
MOVL C01028 V=800.0 PL=0
MOVL C01029 V=800.0 PL=0
MOVL C01030 V=800.0 PL=0
MOVL C01031 V=800.0 PL=0
MOVL C01032 V=800.0 PL=0
MOVL C01033 V=800.0 PL=0
MOVL C01034 V=800.0 PL=0
MOVL C01035 V=800.0 PL=0
MOVL C01036 V=800.0 PL=0
MOVL C01037 V=800.0 PL=0
MOVL C01038 V=800.0 PL=0
MOVL C01039 V=800.0 PL=0
MOVL C01040 V=800.0 PL=0
MOVL C01041 V=800.0 PL=0
MOVL C01042 V=800.0 PL=0
MOVL C01043 V=800.0 PL=0
MOVL C01044 V=800.0 PL=0
MOVL C01045 V=800.0 PL=0
MOVL C01046 V=800.0 PL=0
MOVL C01047 V=800.0 PL=0
MOVL C01048 V=800.0 PL=0
MOVL C01049 V=800.0 PL=0
MOVL C01050 V=800.0 PL=0
MOVL C01051 V=800.0 PL=0
MOVL C01052 V=800.0 PL=0
MOVL C01053 V=800.0 PL=0
MOVL C01054 V=800.0 PL=0
MOVL C01055 V=800.0 PL=0
MOVL C01056 V=800.0 PL=0
MOVL C01057 V=800.0 PL=0
MOVL C01058 V=800.0 PL=0
MOVL C01059 V=800.0 PL=0
MOVL C01060 V=800.0 PL=0
MOVL C01061 V=800.0 PL=0
MOVL C01062 V=800.0 PL=0
MOVL C01063 V=800.0 PL=0
MOVL C01064 V=800.0 PL=0
MOVL C01065 V=800.0 PL=0
MOVL C01066 V=800.0 PL=0
MOVL C01067 V=800.0 PL=0
MOVL C01068 V=800.0 PL=0
MOVL C01069 V=800.0 PL=0
MOVL C01070 V=800.0 PL=0
MOVL C01071 V=800.0 PL=0
MOVL C01072 V=800.0 PL=0
MOVL C01073 V=800.0 PL=0
MOVL C01074 V=800.0 PL=0
MOVL C01075 V=800.0 PL=0
MOVL C01076 V=800.0 PL=0
MOVL C01077 V=800.0 PL=0
MOVL C01078 V=800.0 PL=0
MOVL C01079 V=800.0 PL=0
MOVL C01080 V=800.0 PL=0
MOVL C01081 V=800.0 PL=0
MOVL C01082 V=800.0 PL=0
MOVL C01083 V=800.0 PL=0
MOVL C01084 V=800.0 PL=0
MOVL C01085 V=800.0 PL=0
MOVL C01086 V=800.0 PL=0
MOVL C01087 V=800.0 PL=0
MOVL C01088 V=800.0 PL=0
MOVL C01089 V=800.0 PL=0
MOVL C01090 V=800.0 PL=0
MOVL C01091 V=800.0 PL=0
MOVL C01092 V=800.0 PL=0
MOVL C01093 V=800.0 PL=0
MOVL C01094 V=800.0 PL=0
MOVL C01095 V=800.0 PL=0
MOVL C01096 V=800.0 PL=0
MOVL C01097 V=800.0 PL=0
MOVL C01098 V=800.0 PL=0
MOVL C01099 V=800.0 PL=0
MOVL C01100 V=800.0 PL=0
MOVL C01101 V=800.0 PL=0
MOVL C01102 V=800.0 PL=0
MOVL C01103 V=800.0 PL=0
MOVL C01104 V=800.0 PL=0
MOVL C01105 V=800.0 PL=0
MOVL C01106 V=800.0 PL=0
MOVL C01107 V=800.0 PL=0
MOVL C01108 V=800.0 PL=0
MOVL C01109 V=800.0 PL=0
MOVL C01110 V=800.0 PL=0
MOVL C01111 V=800.0 PL=0
MOVL C01112 V=800.0 PL=0
MOVL C01113 V=800.0 PL=0
MOVL C01114 V=800.0 PL=0
MOVL C01115 V=800.0 PL=0
MOVL C01116 V=800.0 PL=0
MOVL C01117 V=800.0 PL=0
MOVL C01118 V=800.0 PL=0
MOVL C01119 V=800.0 PL=0
MOVL C01120 V=800.0 PL=0
MOVL C01121 V=800.0 PL=0
MOVL C01122 V=800.0 PL=0
MOVL C01123 V=800.0 PL=0
MOVL C01124 V=800.0 PL=0
MOVL C01125 V=800.0 PL=0
MOVL C01126 V=800.0 PL=0
MOVL C01127 V=800.0 PL=0
MOVL C01128 V=800.0 PL=0
MOVL C01129 V=800.0 PL=0
MOVL C01130 V=800.0 PL=0
MOVL C01131 V=800.0 PL=0
MOVL C01132 V=800.0 PL=0
MOVL C01133 V=800.0 PL=0
MOVL C01134 V=800.0 PL=0
MOVL C01135 V=800.0 PL=0
MOVL C01136 V=800.0 PL=0
MOVL C01137 V=800.0 PL=0
MOVL C01138 V=800.0 PL=0
MOVL C01139 V=800.0 PL=0
MOVL C01140 V=800.0 PL=0
MOVL C01141 V=800.0 PL=0
MOVL C01142 V=800.0 PL=0
MOVL C01143 V=800.0 PL=0
MOVL C01144 V=800.0 PL=0
MOVL C01145 V=800.0 PL=0
MOVL C01146 V=800.0 PL=0
MOVL C01147 V=800.0 PL=0
MOVL C01148 V=800.0 PL=0
MOVL C01149 V=800.0 PL=0
MOVL C01150 V=800.0 PL=0
MOVL C01151 V=800.0 PL=0
MOVL C01152 V=800.0 PL=0
MOVL C01153 V=800.0 PL=0
MOVL C01154 V=800.0 PL=0
MOVL C01155 V=800.0 PL=0
MOVL C01156 V=800.0 PL=0
MOVL C01157 V=800.0 PL=0
MOVL C01158 V=800.0 PL=0
MOVL C01159 V=800.0 PL=0
MOVL C01160 V=800.0 PL=0
MOVL C01161 V=800.0 PL=0
MOVL C01162 V=800.0 PL=0
MOVL C01163 V=800.0 PL=0
MOVL C01164 V=800.0 PL=0
MOVL C01165 V=800.0 PL=0
MOVL C01166 V=800.0 PL=0
MOVL C01167 V=800.0 PL=0
MOVL C01168 V=800.0 PL=0
MOVL C01169 V=800.0 PL=0
MOVL C01170 V=800.0 PL=0
MOVL C01171 V=800.0 PL=0
MOVL C01172 V=800.0 PL=0
MOVL C01173 V=800.0 PL=0
MOVL C01174 V=800.0 PL=0
MOVL C01175 V=800.0 PL=0
MOVL C01176 V=800.0 PL=0
MOVL C01177 V=800.0 PL=0
MOVL C01178 V=800.0 PL=0
MOVL C01179 V=800.0 PL=0
MOVL C01180 V=800.0 PL=0
MOVL C01181 V=800.0 PL=0
MOVL C01182 V=800.0 PL=0
MOVL C01183 V=800.0 PL=0
MOVL C01184 V=800.0 PL=0
MOVL C01185 V=800.0 PL=0
MOVL C01186 V=800.0 PL=0
MOVL C01187 V=800.0 PL=0
MOVL C01188 V=800.0 PL=0
MOVL C01189 V=800.0 PL=0
MOVL C01190 V=800.0 PL=0
MOVL C01191 V=800.0 PL=0
MOVL C01192 V=800.0 PL=0
MOVL C01193 V=800.0 PL=0
MOVL C01194 V=800.0 PL=0
MOVL C01195 V=800.0 PL=0
MOVL C01196 V=800.0 PL=0
MOVL C01197 V=800.0 PL=0
MOVL C01198 V=800.0 PL=0
MOVL C01199 V=800.0 PL=0
MOVL C01200 V=800.0 PL=0
MOVL C01201 V=800.0 PL=0
MOVL C01202 V=800.0 PL=0
MOVL C01203 V=800.0 PL=0
MOVL C01204 V=800.0 PL=0
MOVL C01205 V=800.0 PL=0
MOVL C01206 V=800.0 PL=0
MOVL C01207 V=800.0 PL=0
MOVL C01208 V=800.0 PL=0
MOVL C01209 V=800.0 PL=0
MOVL C01210 V=800.0 PL=0
MOVL C01211 V=800.0 PL=0
MOVL C01212 V=800.0 PL=0
MOVL C01213 V=800.0 PL=0
MOVL C01214 V=800.0 PL=0
MOVL C01215 V=800.0 PL=0
MOVL C01216 V=800.0 PL=0
MOVL C01217 V=800.0 PL=0
MOVL C01218 V=800.0 PL=0
MOVL C01219 V=800.0 PL=0
MOVL C01220 V=800.0 PL=0
MOVL C01221 V=800.0 PL=0
MOVL C01222 V=800.0 PL=0
MOVL C01223 V=800.0 PL=0
MOVL C01224 V=800.0 PL=0
MOVL C01225 V=800.0 PL=0
MOVL C01226 V=800.0 PL=0
MOVL C01227 V=800.0 PL=0
MOVL C01228 V=800.0 PL=0
MOVL C01229 V=800.0 PL=0
MOVL C01230 V=800.0 PL=0
MOVL C01231 V=800.0 PL=0
MOVL C01232 V=800.0 PL=0
MOVL C01233 V=800.0 PL=0
MOVL C01234 V=800.0 PL=0
MOVL C01235 V=800.0 PL=0
MOVL C01236 V=800.0 PL=0
MOVL C01237 V=800.0 PL=0
MOVL C01238 V=800.0 PL=0
MOVL C01239 V=800.0 PL=0
MOVL C01240 V=800.0 PL=0
MOVL C01241 V=800.0 PL=0
MOVL C01242 V=800.0 PL=0
MOVL C01243 V=800.0 PL=0
MOVL C01244 V=800.0 PL=0
MOVL C01245 V=800.0 PL=0
MOVL C01246 V=800.0 PL=0
MOVL C01247 V=800.0 PL=0
MOVL C01248 V=800.0 PL=0
MOVL C01249 V=800.0 PL=0
MOVL C01250 V=800.0 PL=0
MOVL C01251 V=800.0 PL=0
MOVL C01252 V=800.0 PL=0
MOVL C01253 V=800.0 PL=0
MOVL C01254 V=800.0 PL=0
MOVL C01255 V=800.0 PL=0
MOVL C01256 V=800.0 PL=0
MOVL C01257 V=800.0 PL=0
MOVL C01258 V=800.0 PL=0
MOVL C01259 V=800.0 PL=0
MOVL C01260 V=800.0 PL=0
MOVL C01261 V=800.0 PL=0
MOVL C01262 V=800.0 PL=0
MOVL C01263 V=800.0 PL=0
MOVL C01264 V=800.0 PL=0
MOVL C01265 V=800.0 PL=0
MOVL C01266 V=800.0 PL=0
MOVL C01267 V=800.0 PL=0
MOVL C01268 V=800.0 PL=0
MOVL C01269 V=800.0 PL=0
MOVL C01270 V=800.0 PL=0
MOVL C01271 V=800.0 PL=0
MOVL C01272 V=800.0 PL=0
MOVL C01273 V=800.0 PL=0
MOVL C01274 V=800.0 PL=0
MOVL C01275 V=800.0 PL=0
MOVL C01276 V=800.0 PL=0
MOVL C01277 V=800.0 PL=0
MOVL C01278 V=800.0 PL=0
MOVL C01279 V=800.0 PL=0
MOVL C01280 V=800.0 PL=0
MOVL C01281 V=800.0 PL=0
MOVL C01282 V=800.0 PL=0
MOVL C01283 V=800.0 PL=0
MOVL C01284 V=800.0 PL=0
MOVL C01285 V=800.0 PL=0
MOVL C01286 V=800.0 PL=0
MOVL C01287 V=800.0 PL=0
MOVL C01288 V=800.0 PL=0
MOVL C01289 V=800.0 PL=0
MOVL C01290 V=800.0 PL=0
MOVL C01291 V=800.0 PL=0
MOVL C01292 V=800.0 PL=0
MOVL C01293 V=800.0 PL=0
MOVL C01294 V=800.0 PL=0
MOVL C01295 V=800.0 PL=0
MOVL C01296 V=800.0 PL=0
MOVL C01297 V=800.0 PL=0
MOVL C01298 V=800.0 PL=0
MOVL C01299 V=800.0 PL=0
MOVL C01300 V=800.0 PL=0
MOVL C01301 V=800.0 PL=0
MOVL C01302 V=800.0 PL=0
MOVL C01303 V=800.0 PL=0
MOVL C01304 V=800.0 PL=0
MOVL C01305 V=800.0 PL=0
MOVL C01306 V=800.0 PL=0
MOVL C01307 V=800.0 PL=0
MOVL C01308 V=800.0 PL=0
MOVL C01309 V=800.0 PL=0
MOVL C01310 V=800.0 PL=0
MOVL C01311 V=800.0 PL=0
MOVL C01312 V=800.0 PL=0
MOVL C01313 V=800.0 PL=0
MOVL C01314 V=800.0 PL=0
MOVL C01315 V=800.0 PL=0
MOVL C01316 V=800.0 PL=0
MOVL C01317 V=800.0 PL=0
MOVL C01318 V=800.0 PL=0
MOVL C01319 V=800.0 PL=0
MOVL C01320 V=800.0 PL=0
MOVL C01321 V=800.0 PL=0
MOVL C01322 V=800.0 PL=0
MOVL C01323 V=800.0 PL=0
MOVL C01324 V=800.0 PL=0
MOVL C01325 V=800.0 PL=0
MOVL C01326 V=800.0 PL=0
MOVL C01327 V=800.0 PL=0
MOVL C01328 V=800.0 PL=0
MOVL C01329 V=800.0 PL=0
MOVL C01330 V=800.0 PL=0
MOVL C01331 V=800.0 PL=0
MOVL C01332 V=800.0 PL=0
MOVL C01333 V=800.0 PL=0
MOVL C01334 V=800.0 PL=0
MOVL C01335 V=800.0 PL=0
MOVL C01336 V=800.0 PL=0
MOVL C01337 V=800.0 PL=0
MOVL C01338 V=800.0 PL=0
MOVL C01339 V=800.0 PL=0
MOVL C01340 V=800.0 PL=0
MOVL C01341 V=800.0 PL=0
MOVL C01342 V=800.0 PL=0
MOVL C01343 V=800.0 PL=0
MOVL C01344 V=800.0 PL=0
MOVL C01345 V=800.0 PL=0
MOVL C01346 V=800.0 PL=0
MOVL C01347 V=800.0 PL=0
MOVL C01348 V=800.0 PL=0
MOVL C01349 V=800.0 PL=0
MOVL C01350 V=800.0 PL=0
MOVL C01351 V=800.0 PL=0
MOVL C01352 V=800.0 PL=0
MOVL C01353 V=800.0 PL=0
MOVL C01354 V=800.0 PL=0
MOVL C01355 V=800.0 PL=0
MOVL C01356 V=800.0 PL=0
MOVL C01357 V=800.0 PL=0
MOVL C01358 V=800.0 PL=0
MOVL C01359 V=800.0 PL=0
MOVL C01360 V=800.0 PL=0
MOVL C01361 V=800.0 PL=0
MOVL C01362 V=800.0 PL=0
MOVL C01363 V=800.0 PL=0
MOVL C01364 V=800.0 PL=0
MOVL C01365 V=800.0 PL=0
MOVL C01366 V=800.0 PL=0
MOVL C01367 V=800.0 PL=0
MOVL C01368 V=800.0 PL=0
MOVL C01369 V=800.0 PL=0
MOVL C01370 V=800.0 PL=0
MOVL C01371 V=800.0 PL=0
MOVL C01372 V=800.0 PL=0
MOVL C01373 V=800.0 PL=0
MOVL C01374 V=800.0 PL=0
MOVL C01375 V=800.0 PL=0
MOVL C01376 V=800.0 PL=0
MOVL C01377 V=800.0 PL=0
MOVL C01378 V=800.0 PL=0
MOVL C01379 V=800.0 PL=0
MOVL C01380 V=800.0 PL=0
MOVL C01381 V=800.0 PL=0
MOVL C01382 V=800.0 PL=0
MOVL C01383 V=800.0 PL=0
MOVL C01384 V=800.0 PL=0
MOVL C01385 V=800.0 PL=0
MOVL C01386 V=800.0 PL=0
MOVL C01387 V=800.0 PL=0
MOVL C01388 V=800.0 PL=0
MOVL C01389 V=800.0 PL=0
MOVL C01390 V=800.0 PL=0
MOVL C01391 V=800.0 PL=0
MOVL C01392 V=800.0 PL=0
MOVL C01393 V=800.0 PL=0
MOVL C01394 V=800.0 PL=0
MOVL C01395 V=800.0 PL=0
MOVL C01396 V=800.0 PL=0
MOVL C01397 V=800.0 PL=0
MOVL C01398 V=800.0 PL=0
MOVL C01399 V=800.0 PL=0
MOVL C01400 V=800.0 PL=0
MOVL C01401 V=800.0 PL=0
MOVL C01402 V=800.0 PL=0
MOVL C01403 V=800.0 PL=0
MOVL C01404 V=800.0 PL=0
MOVL C01405 V=800.0 PL=0
MOVL C01406 V=800.0 PL=0
MOVL C01407 V=800.0 PL=0
MOVL C01408 V=800.0 PL=0
MOVL C01409 V=800.0 PL=0
MOVL C01410 V=800.0 PL=0
MOVL C01411 V=800.0 PL=0
MOVL C01412 V=800.0 PL=0
MOVL C01413 V=800.0 PL=0
MOVL C01414 V=800.0 PL=0
MOVL C01415 V=800.0 PL=0
MOVL C01416 V=800.0 PL=0
MOVL C01417 V=800.0 PL=0
MOVL C01418 V=800.0 PL=0
MOVL C01419 V=800.0 PL=0
MOVL C01420 V=800.0 PL=0
MOVL C01421 V=800.0 PL=0
MOVL C01422 V=800.0 PL=0
MOVL C01423 V=800.0 PL=0
MOVL C01424 V=800.0 PL=0
MOVL C01425 V=800.0 PL=0
MOVL C01426 V=800.0 PL=0
MOVL C01427 V=800.0 PL=0
MOVL C01428 V=800.0 PL=0
MOVL C01429 V=800.0 PL=0
MOVL C01430 V=800.0 PL=0
MOVL C01431 V=800.0 PL=0
MOVL C01432 V=800.0 PL=0
MOVL C01433 V=800.0 PL=0
MOVL C01434 V=800.0 PL=0
MOVL C01435 V=800.0 PL=0
MOVL C01436 V=800.0 PL=0
MOVL C01437 V=800.0 PL=0
MOVL C01438 V=800.0 PL=0
MOVL C01439 V=800.0 PL=0
MOVL C01440 V=800.0 PL=0
MOVL C01441 V=800.0 PL=0
MOVL C01442 V=800.0 PL=0
MOVL C01443 V=800.0 PL=0
MOVL C01444 V=800.0 PL=0
MOVL C01445 V=800.0 PL=0
MOVL C01446 V=800.0 PL=0
MOVL C01447 V=800.0 PL=0
MOVL C01448 V=800.0 PL=0
MOVL C01449 V=800.0 PL=0
MOVL C01450 V=800.0 PL=0
MOVL C01451 V=800.0 PL=0
MOVL C01452 V=800.0 PL=0
MOVL C01453 V=800.0 PL=0
MOVL C01454 V=800.0 PL=0
MOVL C01455 V=800.0 PL=0
MOVL C01456 V=800.0 PL=0
MOVL C01457 V=800.0 PL=0
MOVL C01458 V=800.0 PL=0
MOVL C01459 V=800.0 PL=0
MOVL C01460 V=800.0 PL=0
MOVL C01461 V=800.0 PL=0
MOVL C01462 V=800.0 PL=0
MOVL C01463 V=800.0 PL=0
MOVL C01464 V=800.0 PL=0
MOVL C01465 V=800.0 PL=0
MOVL C01466 V=800.0 PL=0
MOVL C01467 V=800.0 PL=0
MOVL C01468 V=800.0 PL=0
MOVL C01469 V=800.0 PL=0
MOVL C01470 V=800.0 PL=0
MOVL C01471 V=800.0 PL=0
MOVL C01472 V=800.0 PL=0
MOVL C01473 V=800.0 PL=0
MOVL C01474 V=800.0 PL=0
MOVL C01475 V=800.0 PL=0
MOVL C01476 V=800.0 PL=0
MOVL C01477 V=800.0 PL=0
MOVL C01478 V=800.0 PL=0
MOVL C01479 V=800.0 PL=0
MOVL C01480 V=800.0 PL=0
MOVL C01481 V=800.0 PL=0
MOVL C01482 V=800.0 PL=0
MOVL C01483 V=800.0 PL=0
MOVL C01484 V=800.0 PL=0
MOVL C01485 V=800.0 PL=0
MOVL C01486 V=800.0 PL=0
MOVL C01487 V=800.0 PL=0
MOVL C01488 V=800.0 PL=0
MOVL C01489 V=800.0 PL=0
MOVL C01490 V=800.0 PL=0
MOVL C01491 V=800.0 PL=0
MOVL C01492 V=800.0 PL=0
MOVL C01493 V=800.0 PL=0
MOVL C01494 V=800.0 PL=0
MOVL C01495 V=800.0 PL=0
MOVL C01496 V=800.0 PL=0
MOVL C01497 V=800.0 PL=0
MOVL C01498 V=800.0 PL=0
MOVL C01499 V=800.0 PL=0
MOVL C01500 V=800.0 PL=0
MOVL C01501 V=800.0 PL=0
MOVL C01502 V=800.0 PL=0
MOVL C01503 V=800.0 PL=0
MOVL C01504 V=800.0 PL=0
MOVL C01505 V=800.0 PL=0
MOVL C01506 V=800.0 PL=0
MOVL C01507 V=800.0 PL=0
MOVL C01508 V=800.0 PL=0
MOVL C01509 V=800.0 PL=0
MOVL C01510 V=800.0 PL=0
MOVL C01511 V=800.0 PL=0
MOVL C01512 V=800.0 PL=0
MOVL C01513 V=800.0 PL=0
MOVL C01514 V=800.0 PL=0
MOVL C01515 V=800.0 PL=0
MOVL C01516 V=800.0 PL=0
MOVL C01517 V=800.0 PL=0
MOVL C01518 V=800.0 PL=0
MOVL C01519 V=800.0 PL=0
MOVL C01520 V=800.0 PL=0
MOVL C01521 V=800.0 PL=0
MOVL C01522 V=800.0 PL=0
MOVL C01523 V=800.0 PL=0
MOVL C01524 V=800.0 PL=0
MOVL C01525 V=800.0 PL=0
MOVL C01526 V=800.0 PL=0
MOVL C01527 V=800.0 PL=0
MOVL C01528 V=800.0 PL=0
MOVL C01529 V=800.0 PL=0
MOVL C01530 V=800.0 PL=0
MOVL C01531 V=800.0 PL=0
MOVL C01532 V=800.0 PL=0
MOVL C01533 V=800.0 PL=0
MOVL C01534 V=800.0 PL=0
MOVL C01535 V=800.0 PL=0
MOVL C01536 V=800.0 PL=0
MOVL C01537 V=800.0 PL=0
MOVL C01538 V=800.0 PL=0
MOVL C01539 V=800.0 PL=0
MOVL C01540 V=800.0 PL=0
MOVL C01541 V=800.0 PL=0
MOVL C01542 V=800.0 PL=0
MOVL C01543 V=800.0 PL=0
MOVL C01544 V=800.0 PL=0
MOVL C01545 V=800.0 PL=0
MOVL C01546 V=800.0 PL=0
MOVL C01547 V=800.0 PL=0
MOVL C01548 V=800.0 PL=0
MOVL C01549 V=800.0 PL=0
MOVL C01550 V=800.0 PL=0
MOVL C01551 V=800.0 PL=0
MOVL C01552 V=800.0 PL=0
MOVL C01553 V=800.0 PL=0
MOVL C01554 V=800.0 PL=0
MOVL C01555 V=800.0 PL=0
MOVL C01556 V=800.0 PL=0
MOVL C01557 V=800.0 PL=0
MOVL C01558 V=800.0 PL=0
MOVL C01559 V=800.0 PL=0
MOVL C01560 V=800.0 PL=0
MOVL C01561 V=800.0 PL=0
MOVL C01562 V=800.0 PL=0
MOVL C01563 V=800.0 PL=0
MOVL C01564 V=800.0 PL=0
MOVL C01565 V=800.0 PL=0
MOVL C01566 V=800.0 PL=0
MOVL C01567 V=800.0 PL=0
MOVL C01568 V=800.0 PL=0
MOVL C01569 V=800.0 PL=0
MOVL C01570 V=800.0 PL=0
MOVL C01571 V=800.0 PL=0
MOVL C01572 V=800.0 PL=0
MOVL C01573 V=800.0 PL=0
MOVL C01574 V=800.0 PL=0
MOVL C01575 V=800.0 PL=0
MOVL C01576 V=800.0 PL=0
MOVL C01577 V=800.0 PL=0
MOVL C01578 V=800.0 PL=0
MOVL C01579 V=800.0 PL=0
MOVL C01580 V=800.0 PL=0
MOVL C01581 V=800.0 PL=0
MOVL C01582 V=800.0 PL=0
MOVL C01583 V=800.0 PL=0
MOVL C01584 V=800.0 PL=0
MOVL C01585 V=800.0 PL=0
MOVL C01586 V=800.0 PL=0
MOVL C01587 V=800.0 PL=0
MOVL C01588 V=800.0 PL=0
MOVL C01589 V=800.0 PL=0
MOVL C01590 V=800.0 PL=0
MOVL C01591 V=800.0 PL=0
MOVL C01592 V=800.0 PL=0
MOVL C01593 V=800.0 PL=0
MOVL C01594 V=800.0 PL=0
MOVL C01595 V=800.0 PL=0
MOVL C01596 V=800.0 PL=0
MOVL C01597 V=800.0 PL=0
MOVL C01598 V=800.0 PL=0
MOVL C01599 V=800.0 PL=0
MOVL C01600 V=800.0 PL=0
MOVL C01601 V=800.0 PL=0
MOVL C01602 V=800.0 PL=0
MOVL C01603 V=800.0 PL=0
MOVL C01604 V=800.0 PL=0
MOVL C01605 V=800.0 PL=0
MOVL C01606 V=800.0 PL=0
MOVL C01607 V=800.0 PL=0
MOVL C01608 V=800.0 PL=0
MOVL C01609 V=800.0 PL=0
MOVL C01610 V=800.0 PL=0
MOVL C01611 V=800.0 PL=0
MOVL C01612 V=800.0 PL=0
MOVL C01613 V=800.0 PL=0
MOVL C01614 V=800.0 PL=0
MOVL C01615 V=800.0 PL=0
MOVL C01616 V=800.0 PL=0
MOVL C01617 V=800.0 PL=0
MOVL C01618 V=800.0 PL=0
MOVL C01619 V=800.0 PL=0
MOVL C01620 V=800.0 PL=0
MOVL C01621 V=800.0 PL=0
MOVL C01622 V=800.0 PL=0
MOVL C01623 V=800.0 PL=0
MOVL C01624 V=800.0 PL=0
MOVL C01625 V=800.0 PL=0
MOVL C01626 V=800.0 PL=0
MOVL C01627 V=800.0 PL=0
MOVL C01628 V=800.0 PL=0
MOVL C01629 V=800.0 PL=0
MOVL C01630 V=800.0 PL=0
MOVL C01631 V=800.0 PL=0
MOVL C01632 V=800.0 PL=0
MOVL C01633 V=800.0 PL=0
MOVL C01634 V=800.0 PL=0
MOVL C01635 V=800.0 PL=0
MOVL C01636 V=800.0 PL=0
MOVL C01637 V=800.0 PL=0
MOVL C01638 V=800.0 PL=0
MOVL C01639 V=800.0 PL=0
MOVL C01640 V=800.0 PL=0
MOVL C01641 V=800.0 PL=0
MOVL C01642 V=800.0 PL=0
MOVL C01643 V=800.0 PL=0
MOVL C01644 V=800.0 PL=0
MOVL C01645 V=800.0 PL=0
MOVL C01646 V=800.0 PL=0
MOVL C01647 V=800.0 PL=0
MOVL C01648 V=800.0 PL=0
MOVL C01649 V=800.0 PL=0
MOVL C01650 V=800.0 PL=0
MOVL C01651 V=800.0 PL=0
MOVL C01652 V=800.0 PL=0
MOVL C01653 V=800.0 PL=0
MOVL C01654 V=800.0 PL=0
MOVL C01655 V=800.0 PL=0
MOVL C01656 V=800.0 PL=0
MOVL C01657 V=800.0 PL=0
MOVL C01658 V=800.0 PL=0
MOVL C01659 V=800.0 PL=0
MOVL C01660 V=800.0 PL=0
MOVL C01661 V=800.0 PL=0
MOVL C01662 V=800.0 PL=0
MOVL C01663 V=800.0 PL=0
MOVL C01664 V=800.0 PL=0
MOVL C01665 V=800.0 PL=0
MOVL C01666 V=800.0 PL=0
MOVL C01667 V=800.0 PL=0
MOVL C01668 V=800.0 PL=0
MOVL C01669 V=800.0 PL=0
MOVL C01670 V=800.0 PL=0
MOVL C01671 V=800.0 PL=0
MOVL C01672 V=800.0 PL=0
MOVL C01673 V=800.0 PL=0
MOVL C01674 V=800.0 PL=0
MOVL C01675 V=800.0 PL=0
MOVL C01676 V=800.0 PL=0
MOVL C01677 V=800.0 PL=0
MOVL C01678 V=800.0 PL=0
MOVL C01679 V=800.0 PL=0
